// TIA Portal project "AmerikaKamara" (V18)

(* hardware
DEVICE "S7-1200 station_1"  S7-1200 Station
   slot 0: "Rack_0"  S7-1200 Rack  Rack  V1.0
   slot 1: "KamaraFirin"  CPU 1214C DC/DC/DC  6ES7 214-1AG40-0XB0  V4.6
   slot 2: "DI 16/DQ 16x24VDC_1"  6ES7 223-1BL32-0XB0  V2.0
   slot 3: "AQ 4x14BIT_1"  6ES7 232-4HD32-0XB0  V2.1
   slot 3: "CB 1241 (RS485)"  CB 1241 (RS485)  6ES7 241-1CH30-1XB0  V1.0
   slot 4: "AI 4xTC_1"  SM 1231 AI4 x TC  6ES7 231-5QD32-0XB0  V2.0
*)

// ===== PLC "KamaraFirin"  CPU 1214C DC/DC/DC =====

VAR_GLOBAL   // PLC tag table "Default tag table"
   "StartButon" AT %I0.1 : Bool;
   "StopButon" AT %I0.4 : Bool;
   "PompaInvArıza" AT %I0.2 : Bool;
   "ArabaInvArıza" AT %I0.3 : Bool;
   "Tcouple 1" AT %IW128 : Int;
   "Tcouple 1y" AT %IW130 : Int;
   "Tcouple 2" AT %IW132 : Int;
   "Tcouple 2y" AT %IW134 : Int;
   "Damper 1" AT %QW112 : Int;
   "Damper 2" AT %QW114 : Int;
   "Damper 3" AT %QW116 : Int;
   "Damper 4" AT %QW118 : Int;
   "1KapıAcık" AT %I2.0 : Bool;
   "1KapıKapalı" AT %I2.1 : Bool;
   "1KapıYukarda" AT %I2.3 : Bool;
   "1KapıAsagıda" AT %I2.2 : Bool;
   "2KapıAcık" AT %I2.4 : Bool;
   "2KapıKapalı" AT %I2.5 : Bool;
   "2KapıYukarda" AT %I2.7 : Bool;
   "2KapıAsagıda" AT %I2.6 : Bool;
   "1GrupKontaktör" AT %Q2.0 : Bool;
   "1GrupSSR" AT %Q2.1 : Bool;
   "2GrupKontaktör" AT %Q2.4 : Bool;
   "2GrupSSR" AT %Q2.5 : Bool;
   "1KapıAc" AT %Q3.0 : Bool;
   "1KapıKapat" AT %Q3.1 : Bool;
   "1KapıAsagı" AT %Q3.2 : Bool;
   "1KapıYukarı" AT %Q3.3 : Bool;
   "2KapıAc" AT %Q3.4 : Bool;
   "2KapıKapat" AT %Q3.5 : Bool;
   "2KapıAsagı" AT %Q3.6 : Bool;
   "2KapıYukarı" AT %Q3.7 : Bool;
   "AcilStopPano" AT %I0.0 : Bool;
   "HidrolikInverterError" AT %I1.5 : Bool;
   "StartLamba" AT %Q0.0 : Bool;
   "StopLamba" AT %Q0.1 : Bool;
   "HidrolikPompaStart" AT %Q0.2 : Bool;
   "AnaTahliyeValf" AT %Q0.3 : Bool;
   "AcilRöle" AT %Q0.5 : Bool;
   "KırmızıIkaz" AT %Q0.6 : Bool;
   "SarıIkaz" AT %Q0.7 : Bool;
   "YesılIkaz" AT %Q1.0 : Bool;
   "Sıren" AT %Q1.1 : Bool;
   "Emergency" AT %M10.1 : Bool;
   "Error" AT %M10.0 : Bool;
   "currentTemp1Raw" AT %MD100 : Real;
   "currentTemp1" AT %MD104 : Real;
   "SetTimeSnRaw" AT %MD108 : DInt;
   "SetTime" AT %MD112 : Real;
   "SetTemp1Real" AT %MD116 : Real;
   "Ramp1Temp" AT %MD120 : Real;
   "Clock_Byte" AT %MB0 : Byte;
   "Clock_10Hz" AT %M0.0 : Bool;
   "Clock_5Hz" AT %M0.1 : Bool;
   "Clock_2.5Hz" AT %M0.2 : Bool;
   "Clock_2Hz" AT %M0.3 : Bool;
   "Clock_1.25Hz" AT %M0.4 : Bool;
   "Clock_1Hz" AT %M0.5 : Bool;
   "Clock_0.625Hz" AT %M0.6 : Bool;
   "Clock_0.5Hz" AT %M0.7 : Bool;
   "ElapsedSecond" AT %MD124 : Real;
   "elapsed-ramp1" AT %MD128 : Real;
   "StartProcess" AT %M50.0 : Bool;
   "gpwmtimeret1" AT %MD184 : Time;
   "trigclk1" AT %M30.4 : Bool;
   "trigq1" AT %M30.5 : Bool;
   "pwmtimerun1" AT %M30.6 : Bool;
   "pidout1" AT %MD156 : DInt;
   "pidout/20-1" AT %MD188 : UDInt;
   "pidouttime1" AT %MD192 : DWord;
   "currentTemp2Raw" AT %MD160 : Real;
   "currentTemp2" AT %MD164 : Real;
   "SetTemp2Real" AT %MD168 : Real;
   "Ramp2Temp" AT %MD172 : Real;
   "elapsed-ramp2" AT %MD176 : Real;
   "pidout2" AT %MD180 : DInt;
   "trigclk2" AT %M31.0 : Bool;
   "trigq2" AT %M31.1 : Bool;
   "pwmtimerun2" AT %M31.2 : Bool;
   "gpwmtimeret2" AT %MD196 : Time;
   "pidout/20-2" AT %MD200 : UDInt;
   "pidouttime2" AT %MD204 : DWord;
   "Tc1Fark" AT %MD132 : DWord;
   "Tc2Fark" AT %MD136 : DWord;
   "Tc1FarkHata" AT %M30.0 : Bool;
   "Tc2FarkHata" AT %M30.1 : Bool;
   "StepBitti" AT %M30.2 : Bool;
   "StepBittiTrig" AT %M30.3 : Bool;
   "tc1Okunan/10" AT %MD144 : DWord;
   "tc1YOkunan/10" AT %MD148 : DWord;
   "tc2Okunan/10" AT %MD152 : DWord;
   "tc2YOkunan/10" AT %MD140 : DWord;
   "Group2Enable" AT %M20.2 : Bool;
   "Group1Enable" AT %M20.0 : Bool;
   "elapsedTimeTrigClk" AT %M5.0 : Bool;
   "elapsedTimeTrigQ" AT %M5.1 : Bool;
   "startbutonBit" AT %M5.2 : Bool;
   "stopbutonBit" AT %M5.3 : Bool;
   "pidSetTempFark_Q" AT %M5.5 : Bool;
   "baslangicTemp2" AT %MD208 : Real;
   "pidSetTempFark2_Q" AT %M5.6 : Bool;
   "pidSetTemp2" AT %MD212 : Real;
   "baslangicTemp1" AT %MD216 : Real;
   "pidSetTemp1" AT %MD220 : Real;
   "modbusStart" AT %M60.0 : Bool;
   "MBLoadDone" AT %M60.1 : Bool;
   "FrekansCarpilmis" AT %MW224 : UInt;
   "System_Byte" AT %MB1 : Byte;
   "FirstScan" AT %M1.0 : Bool;
   "DiagStatusUpdate" AT %M1.1 : Bool;
   "AlwaysTRUE" AT %M1.2 : Bool;
   "AlwaysFALSE" AT %M1.3 : Bool;
   "ModbusStartScan" AT %M2.0 : Bool;
   "HidrolikBitGeldi" AT %M2.2 : Bool;
   "FrekansYazDone" AT %M60.2 : Bool;
   "KapiAcMinTempError" AT %M350.0 : Bool;
   "DMP1Norm" AT %MD244 : Real;
   "DMP1Scale" AT %MD248 : DWord;
   "DMP2Norm" AT %MD252 : DWord;
   "DMP2Scale" AT %MD256 : DWord;
   "DMP3Norm" AT %MD260 : DWord;
   "DMP3Scale" AT %MD264 : DWord;
   "DMP4Norm" AT %MD268 : DWord;
   "DMP4Scale" AT %MD272 : DWord;
   "HidrolikBit" AT %M400.0 : Bool;
   "akim1Done" AT %M60.4 : Bool;
   "akim2Set" AT %M60.5 : Bool;
   "akim2Done" AT %M60.6 : Bool;
   "akim3Set" AT %M60.7 : Bool;
   "akim1Set" AT %M60.3 : Bool;
   "akim3Done" AT %M61.0 : Bool;
   "akim4Set" AT %M61.1 : Bool;
   "akim4Done" AT %M61.2 : Bool;
   "akim5Set" AT %M61.3 : Bool;
   "akim5Done" AT %M61.4 : Bool;
   "akim6Set" AT %M61.5 : Bool;
   "akim6Done" AT %M61.6 : Bool;
   "HidrolikDelay" AT %MD300 : Time;
   "Tag_1" AT %MD304 : Real;
   "Tag_2" AT %MD308 : DWord;
   "1akim1-2fark" AT %MD312 : DInt;
   "1akim1-2hata" AT %M70.0 : Bool;
   "1akim1-3hata" AT %M70.1 : Bool;
   "1akim1-3fark" AT %MD316 : DInt;
   "1akim2-3fark" AT %MD320 : DInt;
   "1akim2-3hata" AT %M70.2 : Bool;
   "2akim1-2hata" AT %M70.3 : Bool;
   "2akim1-2fark" AT %MD324 : DInt;
   "2akim2-3hata" AT %M70.4 : Bool;
   "2akim1-3fark" AT %MD328 : DInt;
   "2akim2-3hata(1)" AT %M70.5 : Bool;
   "2akim2-3fark" AT %MD332 : DInt;
   "Tag_3" AT %M80.0 : Bool;
   "Reset" AT %M90.0 : Bool;
   "Tag_4" AT %M80.5 : Bool;
   "Tag_5" AT %M5.7 : Bool;
   "kapiacmintemp1" AT %M6.0 : Bool;
   "kapiacmintemp2" AT %M6.1 : Bool;
   "sirenTrigQ" AT %M50.1 : Bool;
   "sirenSet" AT %M50.2 : Bool;
   "kapidelay" AT %MD276 : Time;
   "pompaCalisiyor" AT %M2.3 : Bool;
   "hidrolikdusenkenar" AT %M2.4 : Bool;
END_VAR

DATA_BLOCK "PcdenOkunacak"   // DB2
{ S7_Optimized_Access := 'FALSE' }
VERSION : 0.1
   VAR
      Door1Close : Bool;
      Door1Open : Bool;
      Door1Down : Bool;
      Door1Up : Bool;
      Door2Close : Bool;
      Door2Open : Bool;
      Door2Down : Bool;
      Door2Up : Bool;
      Error : Bool;
      EmergencyPano : Bool;
      HidrolikInveterError : Bool;
      Tc1hata : Bool;
      Tc2Hata : Bool;
      Tc1 : DInt;
      "Tc1.2" : DInt;
      Tc2 : DInt;
      "Tc2.2" : DInt;
      Group1Current : DInt;
      Group2Current : DInt;
      Damper1 : DInt;
      Damper2 : DInt;
      Damper3 : DInt;
      Damper4 : DInt;
      "Step" : DInt;
      butonTime : DInt;
      totalElapsedSec : DInt;
      FirinDurum : Bool;
      butonBasmaTime : Time := T#5S;
      veriGeldi : Bool;
      KapiAcMinTempError : Bool;
      Akim1_1 : Real;
      Akim1_2 : Real;
      Akim1_3 : Real;
      Akim2_1 : Real;
      Akim2_2 : Real;
      Akim2_3 : Real;
      MbLoadError : Bool;
      MbFrekansError : Bool;
      MbAkim1_1Error : Bool;
      MbAkim1_2Error : Bool;
      MbAkim1_3Error : Bool;
      MbAkim2_1Error : Bool;
      MbAkim2_2Error : Bool;
      MbAkim2_3Error : Bool;
      Akim1_1h : Real;
      Akim1_2h : Real;
      Akim1_3h : Real;
      Akim2_1h : Real;
      Akim2_2h : Real;
      Akim2_3h : Real;
      Akim1Ort : DInt;
      Akim2Ort : DInt;
      rezistansError : Bool;
      receteTamam : Bool;
      kapiacildi : Bool;
      Error_1 : Bool;
      siren : Bool;
      elapsedTime : DInt;
      tc1Set : DInt;
      Tc2Set : DInt;
   END_VAR
BEGIN
END_DATA_BLOCK

DATA_BLOCK "PcdenYazilacak"   // DB3
{ S7_Optimized_Access := 'FALSE' }
VERSION : 0.1
   VAR
      Door1Close : Bool;
      Door1Open : Bool;
      Door1Down : Bool;
      Door1Up : Bool;
      Door2Close : Bool;
      Door2Open : Bool;
      Door2Down : Bool;
      Door2Up : Bool;
      SetTemp1 : DInt;
      SetTime : DInt;
      SetTemp2 : DInt;
      Group1Current : DInt;
      Group2Current : DInt;
      Damper1 : DInt;
      Damper2 : DInt;
      Damper3 : DInt;
      Damper4 : DInt;
      TcFarkHata : DInt := 20;
      Group1Run : Bool;
      Group2Run : Bool;
      G1VeriGeldi : Bool;
      G2VeriGeldi : Bool;
      Reset : Bool;
      receteTamam : Bool;
      butonBasmaTime : Time := T#5S;
      SürücüFrekans : Int := 50;
      frekansYaz : Bool;
      sirensustur : Bool;
      MinTemp : DInt := 500;
      ComDelay : Time := T#1s;
      akimFark : DInt := 15;
      adimsayisi : DInt;
   END_VAR
BEGIN
END_DATA_BLOCK

DATA_BLOCK "Group1Control_DB"   // DB6
{ S7_Optimized_Access := 'TRUE' }
VERSION : 0.1
// stored: InstanceOfName Group1Control
"Group1Control"
BEGIN
END_DATA_BLOCK

DATA_BLOCK "Group2Control_DB"   // DB8
{ S7_Optimized_Access := 'TRUE' }
VERSION : 0.1
// stored: InstanceOfName Group2Control
"Group2Control"
BEGIN
END_DATA_BLOCK

// folder: System blocks/Program resources

DATA_BLOCK "ResetTimer"   // DB1
{ S7_Optimized_Access := 'TRUE' }
AUTHOR : Simatic
FAMILY : IEC
NAME : IEC_TMR
VERSION : 1.0
// stored: InstanceOfName IEC_TIMER
"IEC_TIMER"
BEGIN
END_DATA_BLOCK

DATA_BLOCK "IslemBittiTimer"   // DB4
{ S7_Optimized_Access := 'TRUE' }
AUTHOR : Simatic
FAMILY : IEC
NAME : IEC_TMR
VERSION : 1.0
// stored: InstanceOfName IEC_TIMER
"IEC_TIMER"
BEGIN
END_DATA_BLOCK

DATA_BLOCK "Group1PwmTimer"   // DB10
{ S7_Optimized_Access := 'TRUE' }
AUTHOR : Simatic
FAMILY : IEC
NAME : IEC_TMR
VERSION : 1.0
// stored: InstanceOfName IEC_TIMER
"IEC_TIMER"
BEGIN
END_DATA_BLOCK

DATA_BLOCK "Group2PwmTimer"   // DB12
{ S7_Optimized_Access := 'TRUE' }
AUTHOR : Simatic
FAMILY : IEC
NAME : IEC_TMR
VERSION : 1.0
// stored: InstanceOfName IEC_TIMER
"IEC_TIMER"
BEGIN
END_DATA_BLOCK

DATA_BLOCK "AnaValfGecikme"   // DB19
{ S7_Optimized_Access := 'TRUE' }
AUTHOR : Simatic
FAMILY : IEC
NAME : IEC_TMR
VERSION : 1.0
// stored: InstanceOfName IEC_TIMER
"IEC_TIMER"
BEGIN
END_DATA_BLOCK

DATA_BLOCK "PompaGecikme"   // DB20
{ S7_Optimized_Access := 'TRUE' }
AUTHOR : Simatic
FAMILY : IEC
NAME : IEC_TMR
VERSION : 1.0
// stored: InstanceOfName IEC_TIMER
"IEC_TIMER"
BEGIN
END_DATA_BLOCK

DATA_BLOCK "MBCycleDelay"   // DB21
{ S7_Optimized_Access := 'TRUE' }
AUTHOR : Simatic
FAMILY : IEC
NAME : IEC_TMR
VERSION : 1.0
// stored: InstanceOfName IEC_TIMER
"IEC_TIMER"
BEGIN
END_DATA_BLOCK

DATA_BLOCK "akim1TM"   // DB22
{ S7_Optimized_Access := 'TRUE' }
AUTHOR : Simatic
FAMILY : IEC
NAME : IEC_TMR
VERSION : 1.0
// stored: InstanceOfName IEC_TIMER
"IEC_TIMER"
BEGIN
END_DATA_BLOCK

DATA_BLOCK "akim2TM"   // DB23
{ S7_Optimized_Access := 'TRUE' }
AUTHOR : Simatic
FAMILY : IEC
NAME : IEC_TMR
VERSION : 1.0
// stored: InstanceOfName IEC_TIMER
"IEC_TIMER"
BEGIN
END_DATA_BLOCK

DATA_BLOCK "akim3TM"   // DB24
{ S7_Optimized_Access := 'TRUE' }
AUTHOR : Simatic
FAMILY : IEC
NAME : IEC_TMR
VERSION : 1.0
// stored: InstanceOfName IEC_TIMER
"IEC_TIMER"
BEGIN
END_DATA_BLOCK

DATA_BLOCK "akim4TM"   // DB25
{ S7_Optimized_Access := 'TRUE' }
AUTHOR : Simatic
FAMILY : IEC
NAME : IEC_TMR
VERSION : 1.0
// stored: InstanceOfName IEC_TIMER
"IEC_TIMER"
BEGIN
END_DATA_BLOCK

DATA_BLOCK "akim5TM"   // DB26
{ S7_Optimized_Access := 'TRUE' }
AUTHOR : Simatic
FAMILY : IEC
NAME : IEC_TMR
VERSION : 1.0
// stored: InstanceOfName IEC_TIMER
"IEC_TIMER"
BEGIN
END_DATA_BLOCK

DATA_BLOCK "akim6TM"   // DB27
{ S7_Optimized_Access := 'TRUE' }
AUTHOR : Simatic
FAMILY : IEC
NAME : IEC_TMR
VERSION : 1.0
// stored: InstanceOfName IEC_TIMER
"IEC_TIMER"
BEGIN
END_DATA_BLOCK

DATA_BLOCK "IEC_Timer_0_DB"   // DB28
{ S7_Optimized_Access := 'TRUE' }
AUTHOR : Simatic
FAMILY : IEC
NAME : IEC_TMR
VERSION : 1.0
// stored: InstanceOfName IEC_TIMER
"IEC_TIMER"
BEGIN
END_DATA_BLOCK

DATA_BLOCK "rezistansErrorTmr"   // DB29
{ S7_Optimized_Access := 'TRUE' }
AUTHOR : Simatic
FAMILY : IEC
NAME : IEC_TMR
VERSION : 1.0
// stored: InstanceOfName IEC_TIMER
"IEC_TIMER"
BEGIN
END_DATA_BLOCK

DATA_BLOCK "IEC_Timer_0_DB_1"   // DB30
{ S7_Optimized_Access := 'TRUE' }
AUTHOR : Simatic
FAMILY : IEC
NAME : IEC_TMR
VERSION : 1.0
// stored: InstanceOfName IEC_TIMER
"IEC_TIMER"
BEGIN
END_DATA_BLOCK

DATA_BLOCK "IEC_Timer_0_DB_2"   // DB31
{ S7_Optimized_Access := 'TRUE' }
AUTHOR : Simatic
FAMILY : IEC
NAME : IEC_TMR
VERSION : 1.0
// stored: InstanceOfName IEC_TIMER
"IEC_TIMER"
BEGIN
END_DATA_BLOCK

DATA_BLOCK "ErrorStopDelay"   // DB32
{ S7_Optimized_Access := 'TRUE' }
AUTHOR : Simatic
FAMILY : IEC
NAME : IEC_TMR
VERSION : 1.0
// stored: InstanceOfName IEC_TIMER
"IEC_TIMER"
BEGIN
END_DATA_BLOCK

DATA_BLOCK "tcErrorDelay"   // DB33
{ S7_Optimized_Access := 'TRUE' }
AUTHOR : Simatic
FAMILY : IEC
NAME : IEC_TMR
VERSION : 1.0
// stored: InstanceOfName IEC_TIMER
"IEC_TIMER"
BEGIN
END_DATA_BLOCK

DATA_BLOCK "kapi1acikdelay"   // DB35
{ S7_Optimized_Access := 'TRUE' }
AUTHOR : Simatic
FAMILY : IEC
NAME : IEC_TMR
VERSION : 1.0
// stored: InstanceOfName IEC_TIMER
"IEC_TIMER"
BEGIN
END_DATA_BLOCK

DATA_BLOCK "kapi1kapalidelay"   // DB36
{ S7_Optimized_Access := 'TRUE' }
AUTHOR : Simatic
FAMILY : IEC
NAME : IEC_TMR
VERSION : 1.0
// stored: InstanceOfName IEC_TIMER
"IEC_TIMER"
BEGIN
END_DATA_BLOCK

DATA_BLOCK "kapi2acikdelay"   // DB37
{ S7_Optimized_Access := 'TRUE' }
AUTHOR : Simatic
FAMILY : IEC
NAME : IEC_TMR
VERSION : 1.0
// stored: InstanceOfName IEC_TIMER
"IEC_TIMER"
BEGIN
END_DATA_BLOCK

DATA_BLOCK "kapi2kapalidelay"   // DB38
{ S7_Optimized_Access := 'TRUE' }
AUTHOR : Simatic
FAMILY : IEC
NAME : IEC_TMR
VERSION : 1.0
// stored: InstanceOfName IEC_TIMER
"IEC_TIMER"
BEGIN
END_DATA_BLOCK

DATA_BLOCK "sirenSusturtmr"   // DB39
{ S7_Optimized_Access := 'TRUE' }
AUTHOR : Simatic
FAMILY : IEC
NAME : IEC_TMR
VERSION : 1.0
// stored: InstanceOfName IEC_TIMER
"IEC_TIMER"
BEGIN
END_DATA_BLOCK

// folder: (top level)

FUNCTION_BLOCK "Group1Control"   // FB1, LAD
{ S7_Optimized_Access := 'TRUE' }
VERSION : 0.1
   VAR_INPUT
      "m20.0" : Bool;
   END_VAR
BEGIN

REGION Network 1: Group 1 Heating
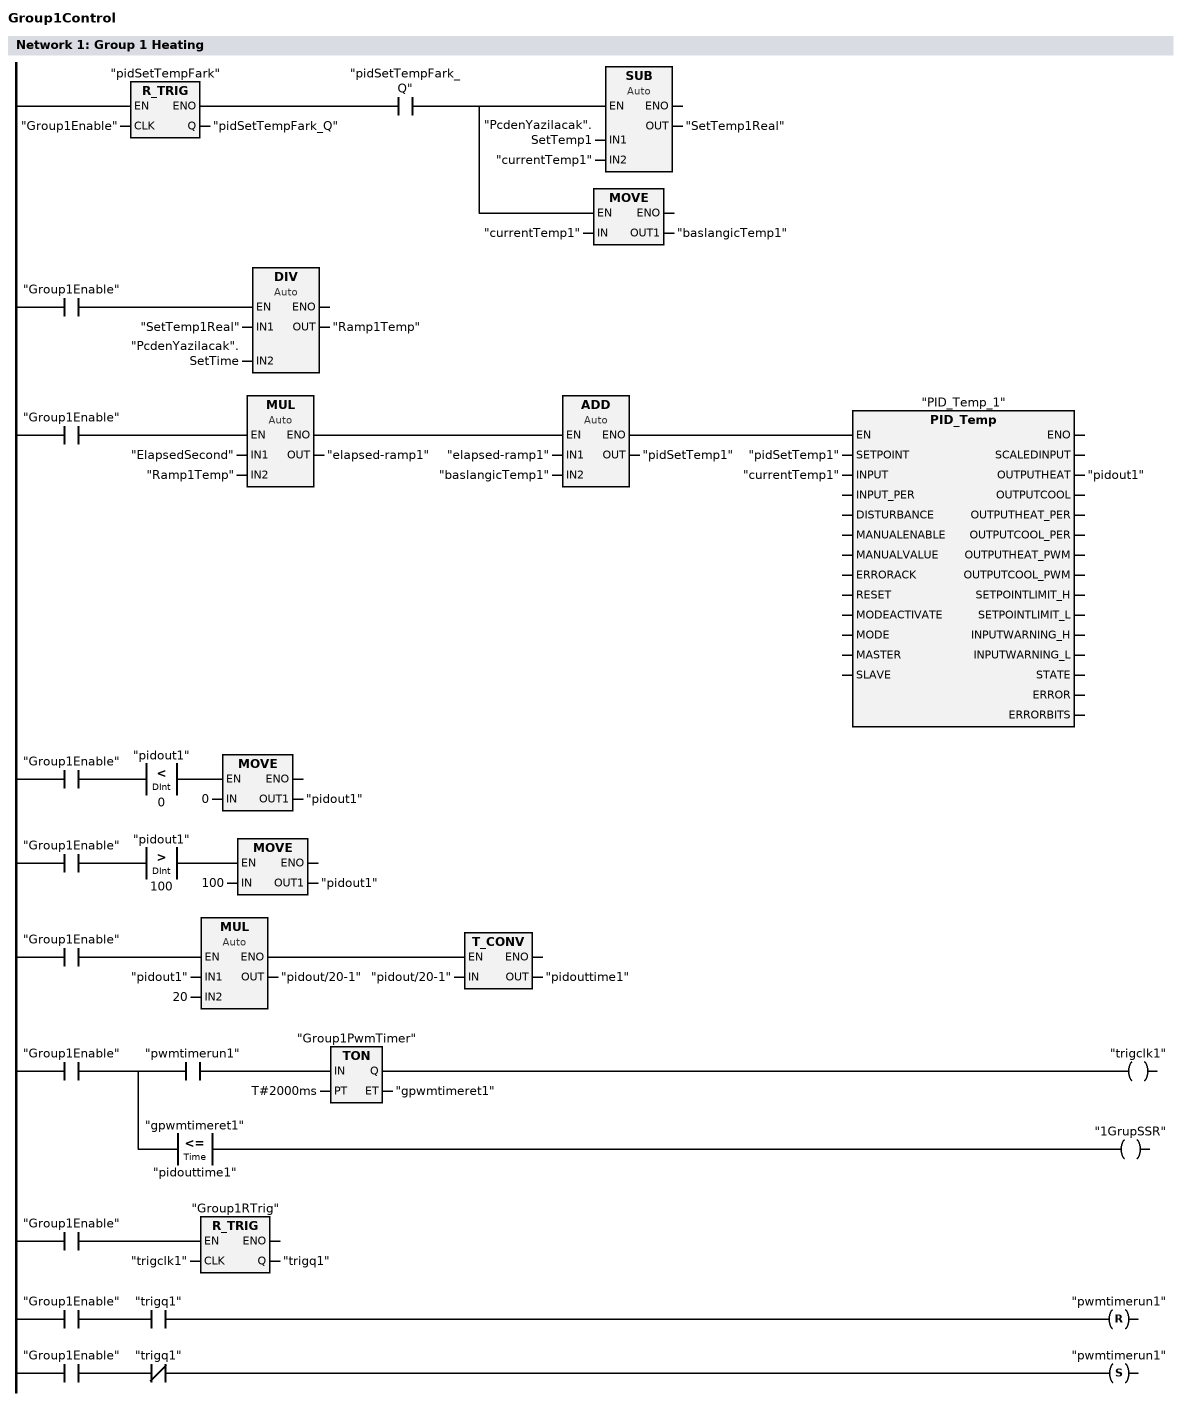
   // ENO of a box is taken as its EN; it also drops when the box reports an error
   "pidSetTempFark"(CLK := "Group1Enable", Q => "pidSetTempFark_Q");   // R_TRIG
   IF "pidSetTempFark_Q" THEN
       "SetTemp1Real" := "PcdenYazilacak".SetTemp1 - "currentTemp1";
       "baslangicTemp1" := "currentTemp1";
   END_IF;
   IF "Group1Enable" THEN
       "Ramp1Temp" := "SetTemp1Real" / "PcdenYazilacak".SetTime;
       "elapsed-ramp1" := "ElapsedSecond" * "Ramp1Temp";
       "pidSetTemp1" := "elapsed-ramp1" + "baslangicTemp1";
       "PID_Temp_1"(Setpoint := "pidSetTemp1", Input := "currentTemp1", OutputHeat => "pidout1");   // PID_Temp
   END_IF;
   IF "Group1Enable" AND ("pidout1" < 0) THEN "pidout1" := 0; END_IF;
   IF "Group1Enable" AND ("pidout1" > 100) THEN "pidout1" := 100; END_IF;
   IF "Group1Enable" THEN
       "pidout/20-1" := "pidout1" * 20;
       "pidouttime1" := T_CONV(IN := "pidout/20-1");
   END_IF;
   "Group1PwmTimer".TON(IN := "Group1Enable" AND "pwmtimerun1", PT := T#2000ms, ET => "gpwmtimeret1");
   "trigclk1" := "Group1PwmTimer".Q;
   "1GrupSSR" := "Group1Enable" AND ("gpwmtimeret1" <= "pidouttime1");
   IF "Group1Enable" THEN
       "Group1RTrig"(CLK := "trigclk1", Q => "trigq1");   // R_TRIG
   END_IF;
   IF "Group1Enable" AND "trigq1" THEN "pwmtimerun1" := FALSE; END_IF;
   IF "Group1Enable" AND NOT "trigq1" THEN "pwmtimerun1" := TRUE; END_IF;
END_REGION
END_FUNCTION_BLOCK

FUNCTION_BLOCK "Group2Control"   // FB2, LAD
{ S7_Optimized_Access := 'TRUE' }
VERSION : 0.1
   VAR_INPUT
      "m20.2" : Bool;
   END_VAR
BEGIN

REGION Network 1
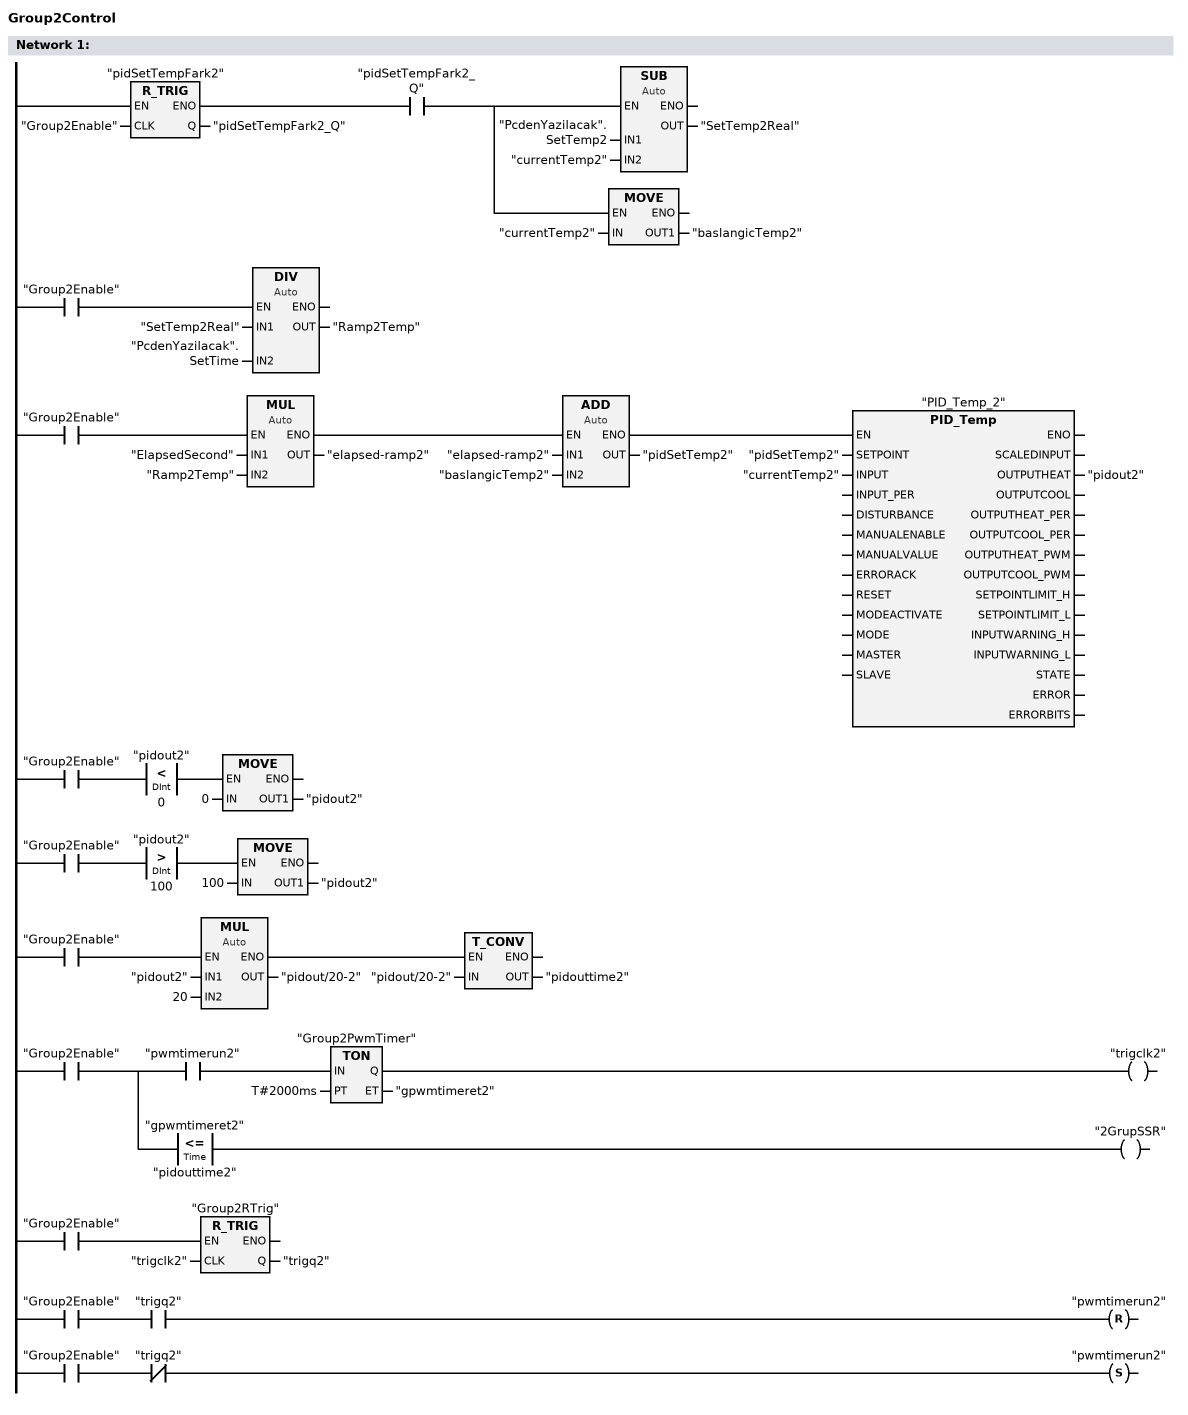
   // ENO of a box is taken as its EN; it also drops when the box reports an error
   "pidSetTempFark2"(CLK := "Group2Enable", Q => "pidSetTempFark2_Q");   // R_TRIG
   IF "pidSetTempFark2_Q" THEN
       "SetTemp2Real" := "PcdenYazilacak".SetTemp2 - "currentTemp2";
       "baslangicTemp2" := "currentTemp2";
   END_IF;
   IF "Group2Enable" THEN
       "Ramp2Temp" := "SetTemp2Real" / "PcdenYazilacak".SetTime;
       "elapsed-ramp2" := "ElapsedSecond" * "Ramp2Temp";
       "pidSetTemp2" := "elapsed-ramp2" + "baslangicTemp2";
       "PID_Temp_2"(Setpoint := "pidSetTemp2", Input := "currentTemp2", OutputHeat => "pidout2");   // PID_Temp
   END_IF;
   IF "Group2Enable" AND ("pidout2" < 0) THEN "pidout2" := 0; END_IF;
   IF "Group2Enable" AND ("pidout2" > 100) THEN "pidout2" := 100; END_IF;
   IF "Group2Enable" THEN
       "pidout/20-2" := "pidout2" * 20;
       "pidouttime2" := T_CONV(IN := "pidout/20-2");
   END_IF;
   "Group2PwmTimer".TON(IN := "Group2Enable" AND "pwmtimerun2", PT := T#2000ms, ET => "gpwmtimeret2");
   "trigclk2" := "Group2PwmTimer".Q;
   "2GrupSSR" := "Group2Enable" AND ("gpwmtimeret2" <= "pidouttime2");
   IF "Group2Enable" THEN
       "Group2RTrig"(CLK := "trigclk2", Q => "trigq2");   // R_TRIG
   END_IF;
   IF "Group2Enable" AND "trigq2" THEN "pwmtimerun2" := FALSE; END_IF;
   IF "Group2Enable" AND NOT "trigq2" THEN "pwmtimerun2" := TRUE; END_IF;
END_REGION
END_FUNCTION_BLOCK

ORGANIZATION_BLOCK "Main"   // OB1, LAD, ProgramCycle
TITLE = "Main Program Sweep (Cycle)"
{ S7_Optimized_Access := 'TRUE' }
VERSION : 0.1
   VAR_INPUT
      Initial_Call : Bool;   // Initial call of this OB
      Remanence : Bool;   // =True, if remanent data are available
   END_VAR
   VAR_TEMP   // added for the SCL form of the ladder/FBD networks
      _w1 : Bool;
      _w2 : Bool;
      _w3 : Bool;
      _w4 : Bool;
      _w5 : Bool;
      _w6 : Bool;
      _w7 : Bool;
   END_VAR
BEGIN

REGION Network 1: startProcess
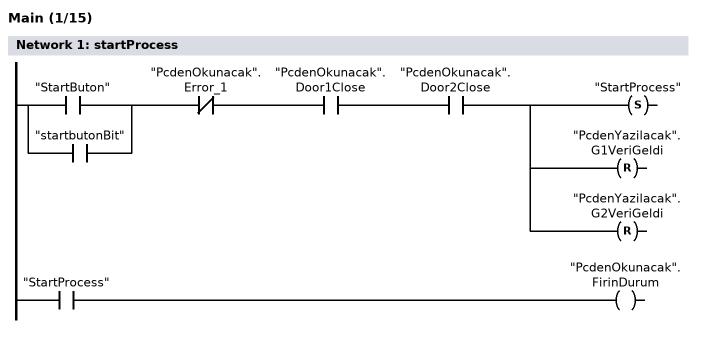
   RUNG wire#powerrail
      Contact( "StartButon" )
      wire#w1
      I_Contact( "PcdenOkunacak".Error_1 )
      Contact( "PcdenOkunacak".Door1Close )
      Contact( "PcdenOkunacak".Door2Close )
      wire#w2
      S_Coil( "StartProcess" )
   END_RUNG
   RUNG wire#powerrail
      Contact( "startbutonBit" )
   END_RUNG wire#w1
   RUNG wire#w2
      R_Coil( "PcdenYazilacak".G1VeriGeldi )
   END_RUNG
   RUNG wire#w2
      R_Coil( "PcdenYazilacak".G2VeriGeldi )
   END_RUNG
   RUNG wire#powerrail
      Contact( "StartProcess" )
      Coil( "PcdenOkunacak".FirinDurum )
   END_RUNG
   // the same network as SCL:
   IF ("StartButon" OR "startbutonBit") AND NOT "PcdenOkunacak".Error_1 AND "PcdenOkunacak".Door1Close AND "PcdenOkunacak".Door2Close THEN
       "StartProcess" := TRUE;
       "PcdenYazilacak".G1VeriGeldi := FALSE;
       "PcdenYazilacak".G2VeriGeldi := FALSE;
   END_IF;
   "PcdenOkunacak".FirinDurum := "StartProcess";
END_REGION

REGION Network 2: Stop and Reset
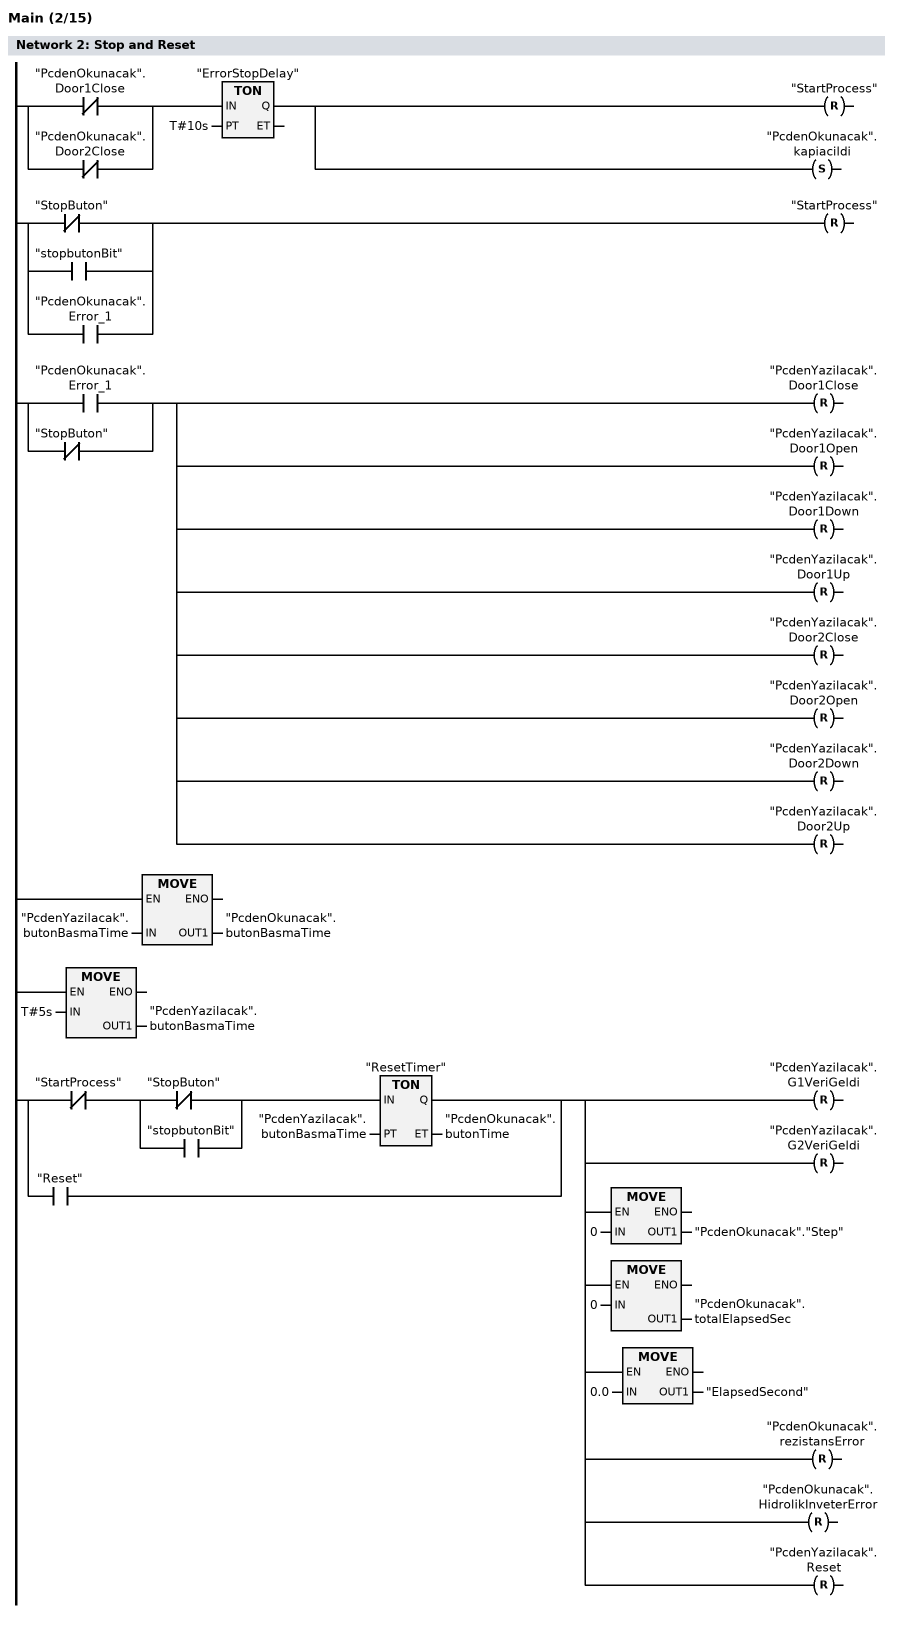
   "ErrorStopDelay".TON(IN := NOT "PcdenOkunacak".Door1Close OR NOT "PcdenOkunacak".Door2Close, PT := T#10s);
   IF "ErrorStopDelay".Q THEN
       "StartProcess" := FALSE;
       "PcdenOkunacak".kapiacildi := TRUE;
   END_IF;
   IF NOT "StopButon" OR "stopbutonBit" OR "PcdenOkunacak".Error_1 THEN "StartProcess" := FALSE; END_IF;
   IF "PcdenOkunacak".Error_1 OR NOT "StopButon" THEN
       "PcdenYazilacak".Door1Close := FALSE;
       "PcdenYazilacak".Door1Open := FALSE;
       "PcdenYazilacak".Door1Down := FALSE;
       "PcdenYazilacak".Door1Up := FALSE;
       "PcdenYazilacak".Door2Close := FALSE;
       "PcdenYazilacak".Door2Open := FALSE;
       "PcdenYazilacak".Door2Down := FALSE;
       "PcdenYazilacak".Door2Up := FALSE;
   END_IF;
   "PcdenOkunacak".butonBasmaTime := "PcdenYazilacak".butonBasmaTime;
   "PcdenYazilacak".butonBasmaTime := T#5s;
   "ResetTimer".TON(IN := NOT "StartProcess" AND (NOT "StopButon" OR "stopbutonBit"),
                    PT := "PcdenYazilacak".butonBasmaTime,
                    ET => "PcdenOkunacak".butonTime);
   IF "ResetTimer".Q OR "Reset" THEN
       "PcdenYazilacak".G1VeriGeldi := FALSE;
       "PcdenYazilacak".G2VeriGeldi := FALSE;
       "PcdenOkunacak"."Step" := 0;
       "PcdenOkunacak".totalElapsedSec := 0;
       "ElapsedSecond" := 0.0;
       "PcdenOkunacak".rezistansError := FALSE;
       "PcdenOkunacak".HidrolikInveterError := FALSE;
       "PcdenYazilacak".Reset := FALSE;
   END_IF;
END_REGION

REGION Network 3: Cycle Step and Time
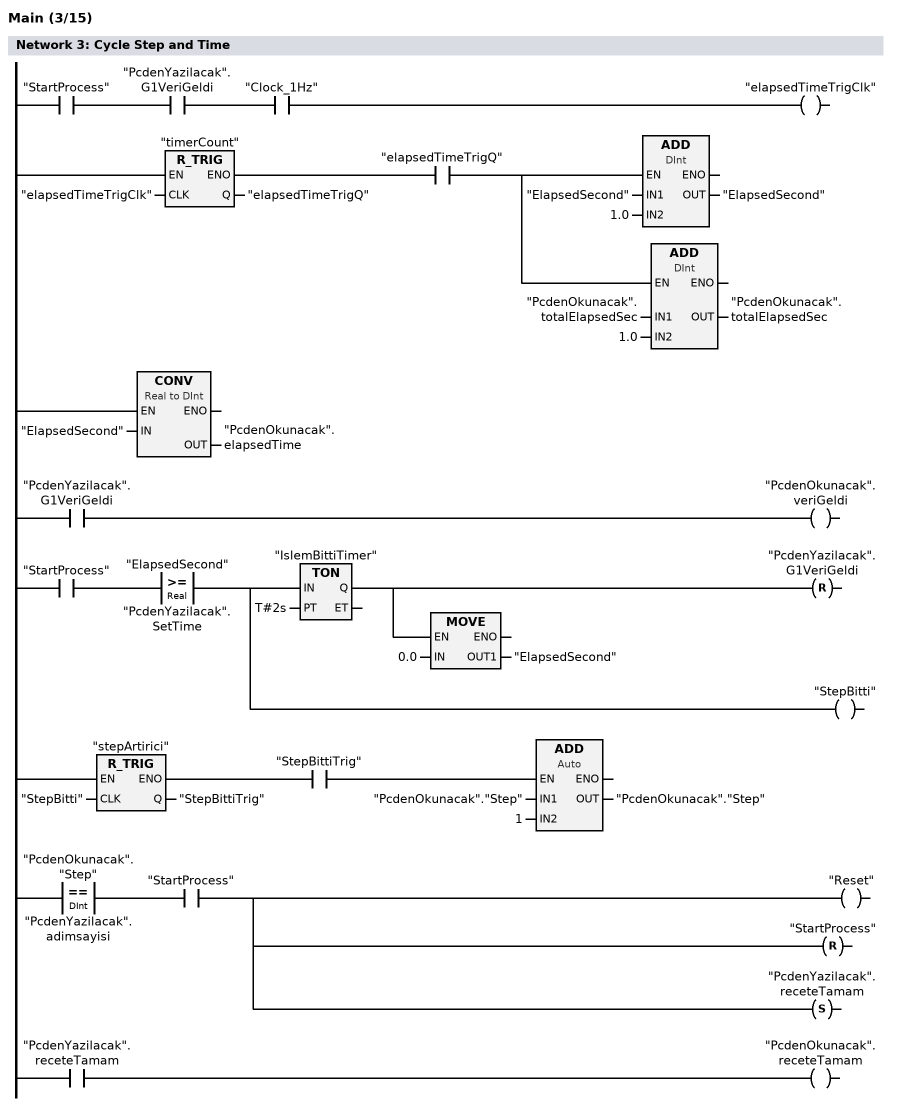
   // ENO of a box is taken as its EN; it also drops when the box reports an error
   "elapsedTimeTrigClk" := "StartProcess" AND "PcdenYazilacak".G1VeriGeldi AND "Clock_1Hz";
   "timerCount"(CLK := "elapsedTimeTrigClk", Q => "elapsedTimeTrigQ");   // R_TRIG
   IF "elapsedTimeTrigQ" THEN
       "ElapsedSecond" := "ElapsedSecond" + 1.0;
       "PcdenOkunacak".totalElapsedSec := "PcdenOkunacak".totalElapsedSec + 1.0;
   END_IF;
   "PcdenOkunacak".elapsedTime := REAL_TO_DINT("ElapsedSecond");
   "PcdenOkunacak".veriGeldi := "PcdenYazilacak".G1VeriGeldi;
   #_w1 := "StartProcess" AND ("ElapsedSecond" >= "PcdenYazilacak".SetTime);
   "IslemBittiTimer".TON(IN := #_w1, PT := T#2s);
   IF "IslemBittiTimer".Q THEN
       "PcdenYazilacak".G1VeriGeldi := FALSE;
       "ElapsedSecond" := 0.0;
   END_IF;
   "StepBitti" := #_w1;
   "stepArtirici"(CLK := "StepBitti", Q => "StepBittiTrig");   // R_TRIG
   IF "StepBittiTrig" THEN "PcdenOkunacak"."Step" := "PcdenOkunacak"."Step" + 1; END_IF;
   "Reset" := ("PcdenOkunacak"."Step" = "PcdenYazilacak".adimsayisi) AND "StartProcess";
   IF "Reset" THEN
       "StartProcess" := FALSE;
       "PcdenYazilacak".receteTamam := TRUE;
   END_IF;
   "PcdenOkunacak".receteTamam := "PcdenYazilacak".receteTamam;
END_REGION

REGION Network 4: Group 1 Heating
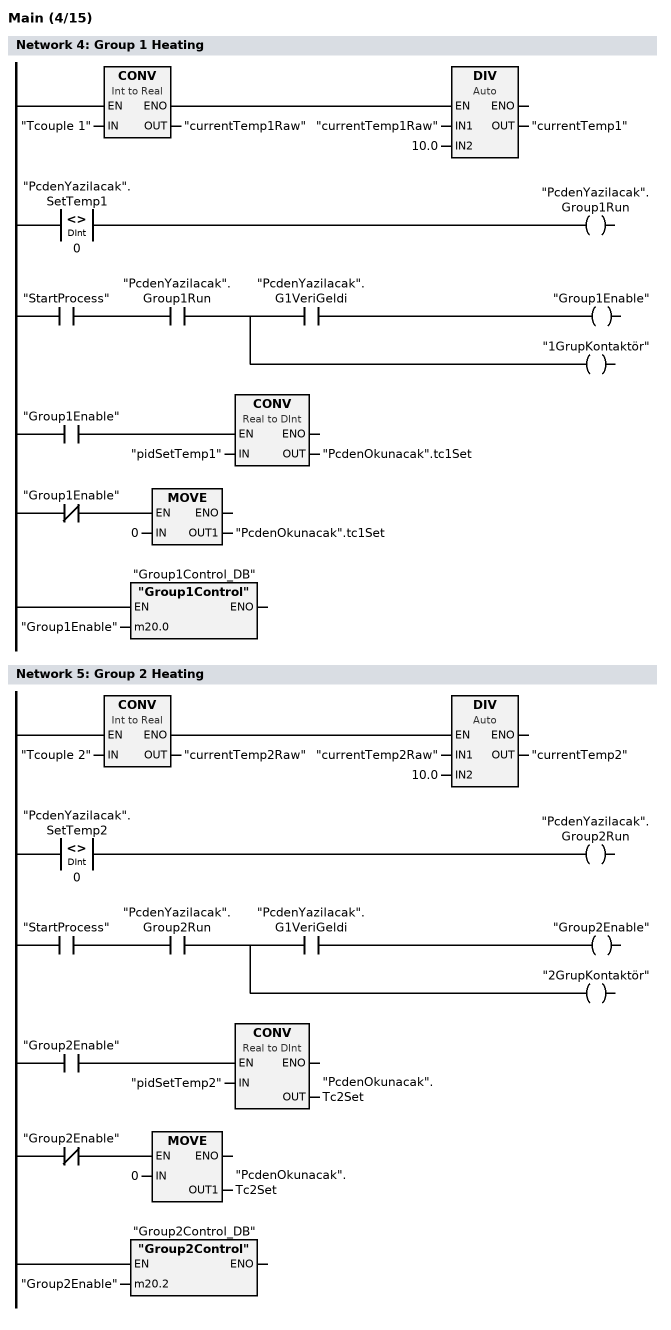
   RUNG wire#powerrail
      { S7_Templates := "[SrcType := Int, DestType := Real]" } Convert(in := "Tcouple 1", out => "currentTemp1Raw")
      Div(in1 := "currentTemp1Raw", in2 := 10.0, out => "currentTemp1")
   END_RUNG
   RUNG wire#powerrail
      { S7_Templates := "SrcType := DInt" } NE_Contact(in1 := "PcdenYazilacak".SetTemp1, in2 := 0)
      Coil( "PcdenYazilacak".Group1Run )
   END_RUNG
   RUNG wire#powerrail
      Contact( "StartProcess" )
      Contact( "PcdenYazilacak".Group1Run )
      wire#w1
      Contact( "PcdenYazilacak".G1VeriGeldi )
      Coil( "Group1Enable" )
   END_RUNG
   RUNG wire#w1
      Coil( "1GrupKontaktör" )
   END_RUNG
   RUNG wire#powerrail
      Contact( "Group1Enable" )
      { S7_Templates := "[SrcType := Real, DestType := DInt]" } Convert(in := "pidSetTemp1", out => "PcdenOkunacak".tc1Set)
   END_RUNG
   RUNG wire#powerrail
      I_Contact( "Group1Enable" )
      Move(in := 0, out1 => "PcdenOkunacak".tc1Set)
   END_RUNG
   RUNG wire#powerrail
      "Group1Control_DB"("m20.0" := "Group1Enable")
   END_RUNG
   // the same network as SCL:
   "currentTemp1Raw" := INT_TO_REAL("Tcouple 1");
   "currentTemp1" := "currentTemp1Raw" / 10.0;
   "PcdenYazilacak".Group1Run := "PcdenYazilacak".SetTemp1 <> 0;
   #_w1 := "StartProcess" AND "PcdenYazilacak".Group1Run;
   "Group1Enable" := #_w1 AND "PcdenYazilacak".G1VeriGeldi;
   "1GrupKontaktör" := #_w1;
   IF "Group1Enable" THEN "PcdenOkunacak".tc1Set := REAL_TO_DINT("pidSetTemp1"); END_IF;
   IF NOT "Group1Enable" THEN "PcdenOkunacak".tc1Set := 0; END_IF;
   "Group1Control_DB"("m20.0" := "Group1Enable");   // "Group1Control"
END_REGION

REGION Network 5: Group 2 Heating
   RUNG wire#powerrail
      { S7_Templates := "[SrcType := Int, DestType := Real]" } Convert(in := "Tcouple 2", out => "currentTemp2Raw")
      Div(in1 := "currentTemp2Raw", in2 := 10.0, out => "currentTemp2")
   END_RUNG
   RUNG wire#powerrail
      { S7_Templates := "SrcType := DInt" } NE_Contact(in1 := "PcdenYazilacak".SetTemp2, in2 := 0)
      Coil( "PcdenYazilacak".Group2Run )
   END_RUNG
   RUNG wire#powerrail
      Contact( "StartProcess" )
      Contact( "PcdenYazilacak".Group2Run )
      wire#w1
      Contact( "PcdenYazilacak".G1VeriGeldi )
      Coil( "Group2Enable" )
   END_RUNG
   RUNG wire#w1
      Coil( "2GrupKontaktör" )
   END_RUNG
   RUNG wire#powerrail
      Contact( "Group2Enable" )
      { S7_Templates := "[SrcType := Real, DestType := DInt]" } Convert(in := "pidSetTemp2", out => "PcdenOkunacak".Tc2Set)
   END_RUNG
   RUNG wire#powerrail
      I_Contact( "Group2Enable" )
      Move(in := 0, out1 => "PcdenOkunacak".Tc2Set)
   END_RUNG
   RUNG wire#powerrail
      "Group2Control_DB"("m20.2" := "Group2Enable")
   END_RUNG
   // the same network as SCL:
   "currentTemp2Raw" := INT_TO_REAL("Tcouple 2");
   "currentTemp2" := "currentTemp2Raw" / 10.0;
   "PcdenYazilacak".Group2Run := "PcdenYazilacak".SetTemp2 <> 0;
   #_w1 := "StartProcess" AND "PcdenYazilacak".Group2Run;
   "Group2Enable" := #_w1 AND "PcdenYazilacak".G1VeriGeldi;
   "2GrupKontaktör" := #_w1;
   IF "Group2Enable" THEN "PcdenOkunacak".Tc2Set := REAL_TO_DINT("pidSetTemp2"); END_IF;
   IF NOT "Group2Enable" THEN "PcdenOkunacak".Tc2Set := 0; END_IF;
   "Group2Control_DB"("m20.2" := "Group2Enable");   // "Group2Control"
END_REGION

REGION Network 6: TCouple
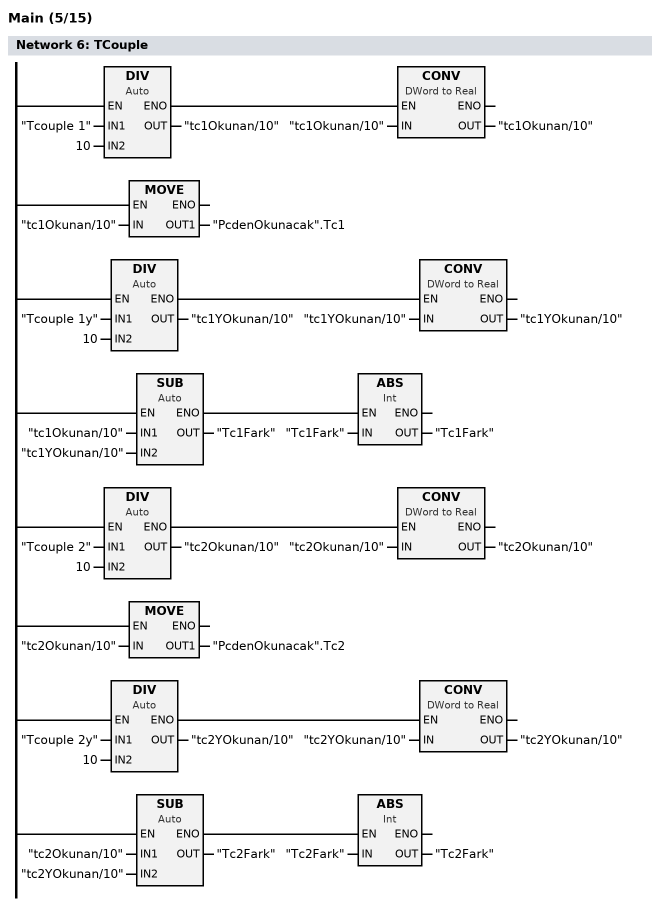
   RUNG wire#powerrail
      Div(in1 := "Tcouple 1", in2 := 10, out => "tc1Okunan/10")
      { S7_Templates := "[SrcType := DWord, DestType := Real]" } Convert(in := "tc1Okunan/10", out => "tc1Okunan/10")
   END_RUNG
   RUNG wire#powerrail
      Move(in := "tc1Okunan/10", out1 => "PcdenOkunacak".Tc1)
   END_RUNG
   RUNG wire#powerrail
      Div(in1 := "Tcouple 1y", in2 := 10, out => "tc1YOkunan/10")
      { S7_Templates := "[SrcType := DWord, DestType := Real]" } Convert(in := "tc1YOkunan/10", out => "tc1YOkunan/10")
   END_RUNG
   RUNG wire#powerrail
      Sub(in1 := "tc1Okunan/10", in2 := "tc1YOkunan/10", out => "Tc1Fark")
      { S7_Templates := "SrcType := Int" } Abs(in := "Tc1Fark", out => "Tc1Fark")
   END_RUNG
   RUNG wire#powerrail
      Div(in1 := "Tcouple 2", in2 := 10, out => "tc2Okunan/10")
      { S7_Templates := "[SrcType := DWord, DestType := Real]" } Convert(in := "tc2Okunan/10", out => "tc2Okunan/10")
   END_RUNG
   RUNG wire#powerrail
      Move(in := "tc2Okunan/10", out1 => "PcdenOkunacak".Tc2)
   END_RUNG
   RUNG wire#powerrail
      Div(in1 := "Tcouple 2y", in2 := 10, out => "tc2YOkunan/10")
      { S7_Templates := "[SrcType := DWord, DestType := Real]" } Convert(in := "tc2YOkunan/10", out => "tc2YOkunan/10")
   END_RUNG
   RUNG wire#powerrail
      Sub(in1 := "tc2Okunan/10", in2 := "tc2YOkunan/10", out => "Tc2Fark")
      { S7_Templates := "SrcType := Int" } Abs(in := "Tc2Fark", out => "Tc2Fark")
   END_RUNG
   // the same network as SCL:
   "tc1Okunan/10" := "Tcouple 1" / 10;
   "tc1Okunan/10" := DWORD_TO_REAL("tc1Okunan/10");
   "PcdenOkunacak".Tc1 := "tc1Okunan/10";
   "tc1YOkunan/10" := "Tcouple 1y" / 10;
   "tc1YOkunan/10" := DWORD_TO_REAL("tc1YOkunan/10");
   "Tc1Fark" := "tc1Okunan/10" - "tc1YOkunan/10";
   "Tc1Fark" := ABS("Tc1Fark");
   "tc2Okunan/10" := "Tcouple 2" / 10;
   "tc2Okunan/10" := DWORD_TO_REAL("tc2Okunan/10");
   "PcdenOkunacak".Tc2 := "tc2Okunan/10";
   "tc2YOkunan/10" := "Tcouple 2y" / 10;
   "tc2YOkunan/10" := DWORD_TO_REAL("tc2YOkunan/10");
   "Tc2Fark" := "tc2Okunan/10" - "tc2YOkunan/10";
   "Tc2Fark" := ABS("Tc2Fark");
END_REGION

REGION Network 7: Emergency
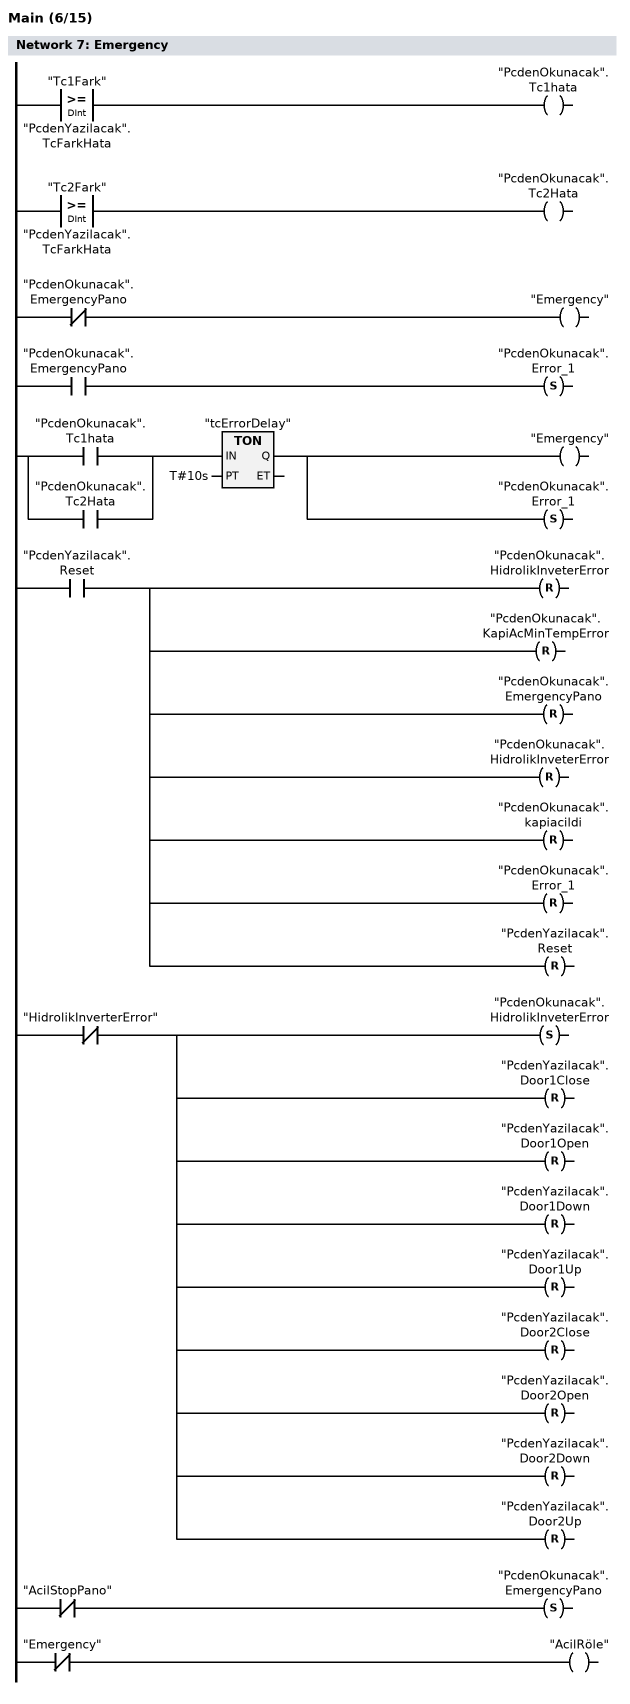
   "PcdenOkunacak".Tc1hata := "Tc1Fark" >= "PcdenYazilacak".TcFarkHata;
   "PcdenOkunacak".Tc2Hata := "Tc2Fark" >= "PcdenYazilacak".TcFarkHata;
   "Emergency" := NOT "PcdenOkunacak".EmergencyPano;
   IF "PcdenOkunacak".EmergencyPano THEN "PcdenOkunacak".Error_1 := TRUE; END_IF;
   "tcErrorDelay".TON(IN := "PcdenOkunacak".Tc1hata OR "PcdenOkunacak".Tc2Hata, PT := T#10s);
   "Emergency" := "tcErrorDelay".Q;
   IF "tcErrorDelay".Q THEN "PcdenOkunacak".Error_1 := TRUE; END_IF;
   IF "PcdenYazilacak".Reset THEN
       "PcdenOkunacak".HidrolikInveterError := FALSE;
       "PcdenOkunacak".KapiAcMinTempError := FALSE;
       "PcdenOkunacak".EmergencyPano := FALSE;
       "PcdenOkunacak".HidrolikInveterError := FALSE;
       "PcdenOkunacak".kapiacildi := FALSE;
       "PcdenOkunacak".Error_1 := FALSE;
       "PcdenYazilacak".Reset := FALSE;
   END_IF;
   IF NOT "HidrolikInverterError" THEN
       "PcdenOkunacak".HidrolikInveterError := TRUE;
       "PcdenYazilacak".Door1Close := FALSE;
       "PcdenYazilacak".Door1Open := FALSE;
       "PcdenYazilacak".Door1Down := FALSE;
       "PcdenYazilacak".Door1Up := FALSE;
       "PcdenYazilacak".Door2Close := FALSE;
       "PcdenYazilacak".Door2Open := FALSE;
       "PcdenYazilacak".Door2Down := FALSE;
       "PcdenYazilacak".Door2Up := FALSE;
   END_IF;
   IF NOT "AcilStopPano" THEN "PcdenOkunacak".EmergencyPano := TRUE; END_IF;
   "AcilRöle" := NOT "Emergency";
END_REGION

REGION Network 8: Door Inputs
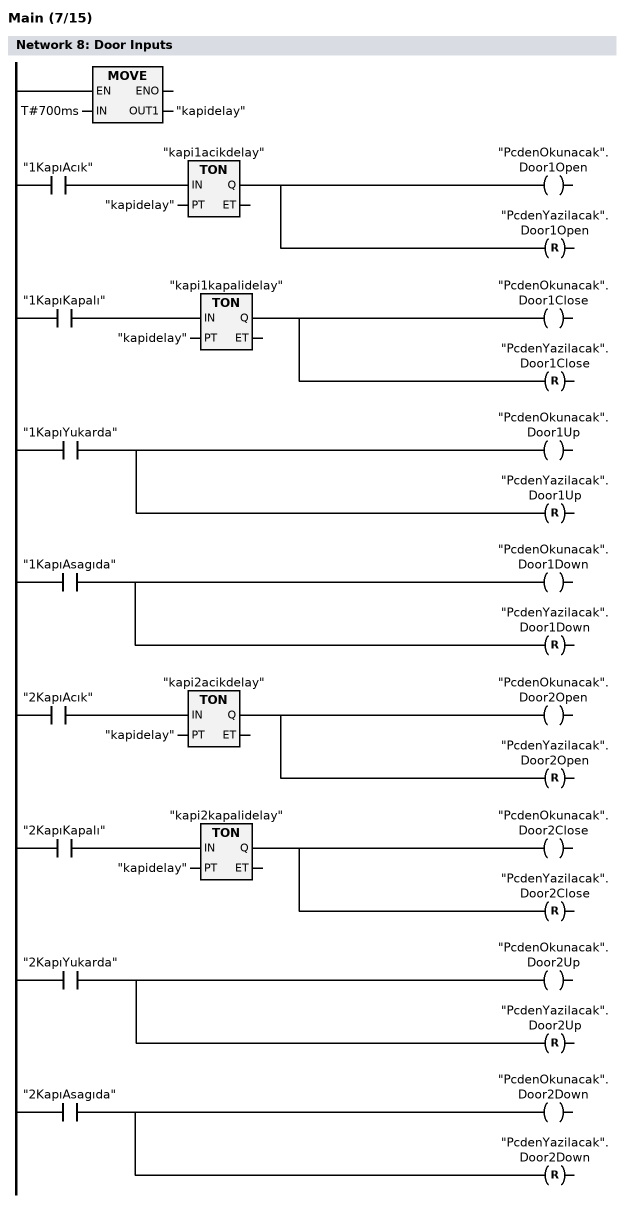
   "kapidelay" := T#700ms;
   "kapi1acikdelay".TON(IN := "1KapıAcık", PT := "kapidelay");
   "PcdenOkunacak".Door1Open := "kapi1acikdelay".Q;
   IF "kapi1acikdelay".Q THEN "PcdenYazilacak".Door1Open := FALSE; END_IF;
   "kapi1kapalidelay".TON(IN := "1KapıKapalı", PT := "kapidelay");
   "PcdenOkunacak".Door1Close := "kapi1kapalidelay".Q;
   IF "kapi1kapalidelay".Q THEN "PcdenYazilacak".Door1Close := FALSE; END_IF;
   "PcdenOkunacak".Door1Up := "1KapıYukarda";
   IF "1KapıYukarda" THEN "PcdenYazilacak".Door1Up := FALSE; END_IF;
   "PcdenOkunacak".Door1Down := "1KapıAsagıda";
   IF "1KapıAsagıda" THEN "PcdenYazilacak".Door1Down := FALSE; END_IF;
   "kapi2acikdelay".TON(IN := "2KapıAcık", PT := "kapidelay");
   "PcdenOkunacak".Door2Open := "kapi2acikdelay".Q;
   IF "kapi2acikdelay".Q THEN "PcdenYazilacak".Door2Open := FALSE; END_IF;
   "kapi2kapalidelay".TON(IN := "2KapıKapalı", PT := "kapidelay");
   "PcdenOkunacak".Door2Close := "kapi2kapalidelay".Q;
   IF "kapi2kapalidelay".Q THEN "PcdenYazilacak".Door2Close := FALSE; END_IF;
   "PcdenOkunacak".Door2Up := "2KapıYukarda";
   IF "2KapıYukarda" THEN "PcdenYazilacak".Door2Up := FALSE; END_IF;
   "PcdenOkunacak".Door2Down := "2KapıAsagıda";
   IF "2KapıAsagıda" THEN "PcdenYazilacak".Door2Down := FALSE; END_IF;
END_REGION

REGION Network 9: Door 1 Outputs
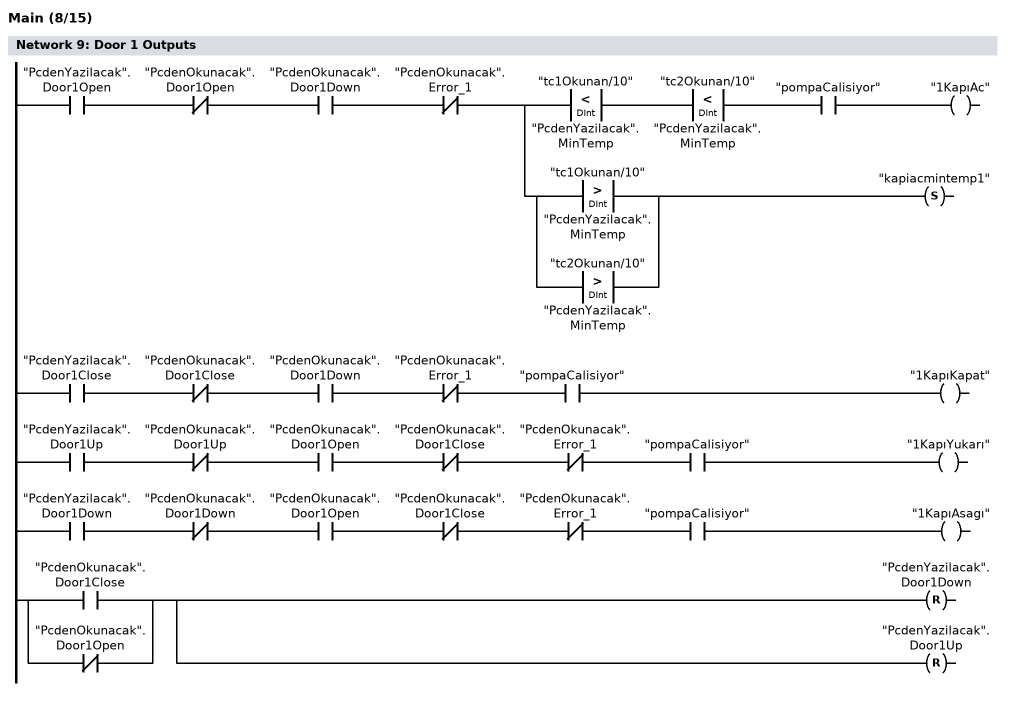
   RUNG wire#powerrail
      Contact( "PcdenYazilacak".Door1Open )
      I_Contact( "PcdenOkunacak".Door1Open )
      Contact( "PcdenOkunacak".Door1Down )
      I_Contact( "PcdenOkunacak".Error_1 )
      wire#w1
      { S7_Templates := "SrcType := DInt" } LT_Contact(in1 := "tc1Okunan/10", in2 := "PcdenYazilacak".MinTemp)
      { S7_Templates := "SrcType := DInt" } LT_Contact(in1 := "tc2Okunan/10", in2 := "PcdenYazilacak".MinTemp)
      Contact( "pompaCalisiyor" )
      Coil( "1KapıAc" )
   END_RUNG
   RUNG wire#w1
      { S7_Templates := "SrcType := DInt" } GT_Contact(in1 := "tc1Okunan/10", in2 := "PcdenYazilacak".MinTemp)
      wire#w2
      S_Coil( "kapiacmintemp1" )
   END_RUNG
   RUNG wire#w1
      { S7_Templates := "SrcType := DInt" } GT_Contact(in1 := "tc2Okunan/10", in2 := "PcdenYazilacak".MinTemp)
   END_RUNG wire#w2
   RUNG wire#powerrail
      Contact( "PcdenYazilacak".Door1Close )
      I_Contact( "PcdenOkunacak".Door1Close )
      Contact( "PcdenOkunacak".Door1Down )
      I_Contact( "PcdenOkunacak".Error_1 )
      Contact( "pompaCalisiyor" )
      Coil( "1KapıKapat" )
   END_RUNG
   RUNG wire#powerrail
      Contact( "PcdenYazilacak".Door1Up )
      I_Contact( "PcdenOkunacak".Door1Up )
      Contact( "PcdenOkunacak".Door1Open )
      I_Contact( "PcdenOkunacak".Door1Close )
      I_Contact( "PcdenOkunacak".Error_1 )
      Contact( "pompaCalisiyor" )
      Coil( "1KapıYukarı" )
   END_RUNG
   RUNG wire#powerrail
      Contact( "PcdenYazilacak".Door1Down )
      I_Contact( "PcdenOkunacak".Door1Down )
      Contact( "PcdenOkunacak".Door1Open )
      I_Contact( "PcdenOkunacak".Door1Close )
      I_Contact( "PcdenOkunacak".Error_1 )
      Contact( "pompaCalisiyor" )
      Coil( "1KapıAsagı" )
   END_RUNG
   RUNG wire#powerrail
      Contact( "PcdenOkunacak".Door1Close )
      wire#w3
      R_Coil( "PcdenYazilacak".Door1Down )
   END_RUNG
   RUNG wire#powerrail
      I_Contact( "PcdenOkunacak".Door1Open )
   END_RUNG wire#w3
   RUNG wire#w3
      R_Coil( "PcdenYazilacak".Door1Up )
   END_RUNG
   // the same network as SCL:
   #_w1 := "PcdenYazilacak".Door1Open AND NOT "PcdenOkunacak".Door1Open AND "PcdenOkunacak".Door1Down AND NOT "PcdenOkunacak".Error_1;
   "1KapıAc" := #_w1 AND ("tc1Okunan/10" < "PcdenYazilacak".MinTemp) AND ("tc2Okunan/10" < "PcdenYazilacak".MinTemp) AND "pompaCalisiyor";
   IF #_w1 AND (("tc1Okunan/10" > "PcdenYazilacak".MinTemp) OR ("tc2Okunan/10" > "PcdenYazilacak".MinTemp)) THEN
       "kapiacmintemp1" := TRUE;
   END_IF;
   "1KapıKapat" := "PcdenYazilacak".Door1Close AND NOT "PcdenOkunacak".Door1Close AND "PcdenOkunacak".Door1Down AND NOT "PcdenOkunacak".Error_1 AND "pompaCalisiyor";
   "1KapıYukarı" := "PcdenYazilacak".Door1Up AND NOT "PcdenOkunacak".Door1Up AND "PcdenOkunacak".Door1Open AND NOT "PcdenOkunacak".Door1Close AND NOT "PcdenOkunacak".Error_1 AND "pompaCalisiyor";
   "1KapıAsagı" := "PcdenYazilacak".Door1Down AND NOT "PcdenOkunacak".Door1Down AND "PcdenOkunacak".Door1Open AND NOT "PcdenOkunacak".Door1Close AND NOT "PcdenOkunacak".Error_1 AND "pompaCalisiyor";
   IF "PcdenOkunacak".Door1Close OR NOT "PcdenOkunacak".Door1Open THEN
       "PcdenYazilacak".Door1Down := FALSE;
       "PcdenYazilacak".Door1Up := FALSE;
   END_IF;
END_REGION

REGION Network 10: Door 2 Outputs
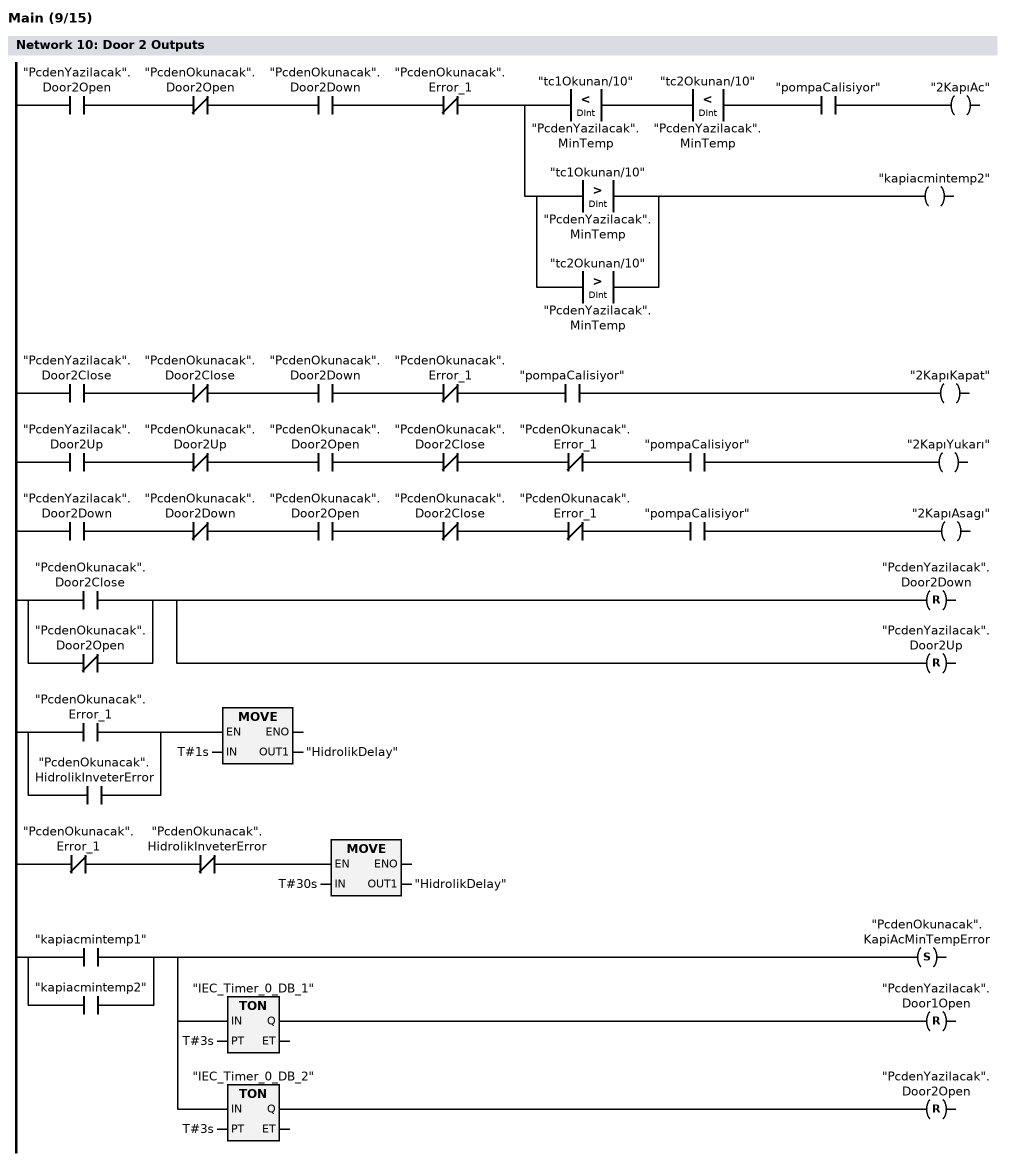
   #_w1 := "PcdenYazilacak".Door2Open AND NOT "PcdenOkunacak".Door2Open AND "PcdenOkunacak".Door2Down AND NOT "PcdenOkunacak".Error_1;
   "2KapıAc" := #_w1 AND ("tc1Okunan/10" < "PcdenYazilacak".MinTemp) AND ("tc2Okunan/10" < "PcdenYazilacak".MinTemp) AND "pompaCalisiyor";
   "kapiacmintemp2" := #_w1 AND (("tc1Okunan/10" > "PcdenYazilacak".MinTemp) OR ("tc2Okunan/10" > "PcdenYazilacak".MinTemp));
   "2KapıKapat" := "PcdenYazilacak".Door2Close AND NOT "PcdenOkunacak".Door2Close AND "PcdenOkunacak".Door2Down AND NOT "PcdenOkunacak".Error_1 AND "pompaCalisiyor";
   "2KapıYukarı" := "PcdenYazilacak".Door2Up AND NOT "PcdenOkunacak".Door2Up AND "PcdenOkunacak".Door2Open AND NOT "PcdenOkunacak".Door2Close AND NOT "PcdenOkunacak".Error_1 AND "pompaCalisiyor";
   "2KapıAsagı" := "PcdenYazilacak".Door2Down AND NOT "PcdenOkunacak".Door2Down AND "PcdenOkunacak".Door2Open AND NOT "PcdenOkunacak".Door2Close AND NOT "PcdenOkunacak".Error_1 AND "pompaCalisiyor";
   IF "PcdenOkunacak".Door2Close OR NOT "PcdenOkunacak".Door2Open THEN
       "PcdenYazilacak".Door2Down := FALSE;
       "PcdenYazilacak".Door2Up := FALSE;
   END_IF;
   IF "PcdenOkunacak".Error_1 OR "PcdenOkunacak".HidrolikInveterError THEN "HidrolikDelay" := T#1s; END_IF;
   IF NOT "PcdenOkunacak".Error_1 AND NOT "PcdenOkunacak".HidrolikInveterError THEN
       "HidrolikDelay" := T#30s;
   END_IF;
   #_w2 := "kapiacmintemp1" OR "kapiacmintemp2";
   IF #_w2 THEN "PcdenOkunacak".KapiAcMinTempError := TRUE; END_IF;
   "IEC_Timer_0_DB_1".TON(IN := #_w2, PT := T#3s);
   IF "IEC_Timer_0_DB_1".Q THEN "PcdenYazilacak".Door1Open := FALSE; END_IF;
   "IEC_Timer_0_DB_2".TON(IN := #_w2, PT := T#3s);
   IF "IEC_Timer_0_DB_2".Q THEN "PcdenYazilacak".Door2Open := FALSE; END_IF;
END_REGION

REGION Network 11: Hidrolik Pompa
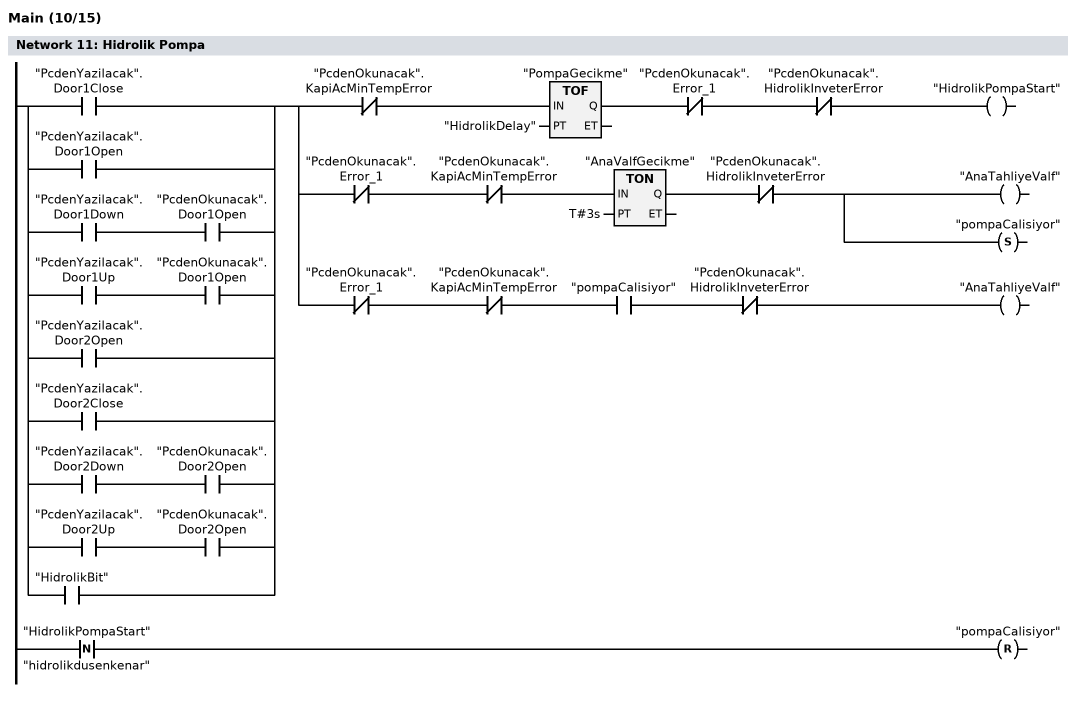
   #_w1 := "PcdenYazilacak".Door1Close OR "PcdenYazilacak".Door1Open OR ("PcdenYazilacak".Door1Down AND "PcdenOkunacak".Door1Open) OR ("PcdenYazilacak".Door1Up AND "PcdenOkunacak".Door1Open) OR "PcdenYazilacak".Door2Open OR "PcdenYazilacak".Door2Close OR ("PcdenYazilacak".Door2Down AND "PcdenOkunacak".Door2Open) OR ("PcdenYazilacak".Door2Up AND "PcdenOkunacak".Door2Open) OR "HidrolikBit";
   "PompaGecikme".TOF(IN := #_w1 AND NOT "PcdenOkunacak".KapiAcMinTempError, PT := "HidrolikDelay");
   "HidrolikPompaStart" := "PompaGecikme".Q AND NOT "PcdenOkunacak".Error_1 AND NOT "PcdenOkunacak".HidrolikInveterError;
   "AnaValfGecikme".TON(IN := #_w1 AND NOT "PcdenOkunacak".Error_1 AND NOT "PcdenOkunacak".KapiAcMinTempError,
                        PT := T#3s);
   "AnaTahliyeValf" := "AnaValfGecikme".Q AND NOT "PcdenOkunacak".HidrolikInveterError;
   IF "AnaTahliyeValf" THEN "pompaCalisiyor" := TRUE; END_IF;
   "AnaTahliyeValf" := #_w1 AND NOT "PcdenOkunacak".Error_1 AND NOT "PcdenOkunacak".KapiAcMinTempError AND "pompaCalisiyor" AND NOT "PcdenOkunacak".HidrolikInveterError;
   #_w2 := NOT "HidrolikPompaStart" AND "hidrolikdusenkenar";   // falling edge of "HidrolikPompaStart"
   "hidrolikdusenkenar" := "HidrolikPompaStart";
   IF #_w2 THEN "pompaCalisiyor" := FALSE; END_IF;
END_REGION

REGION Network 12: Communication
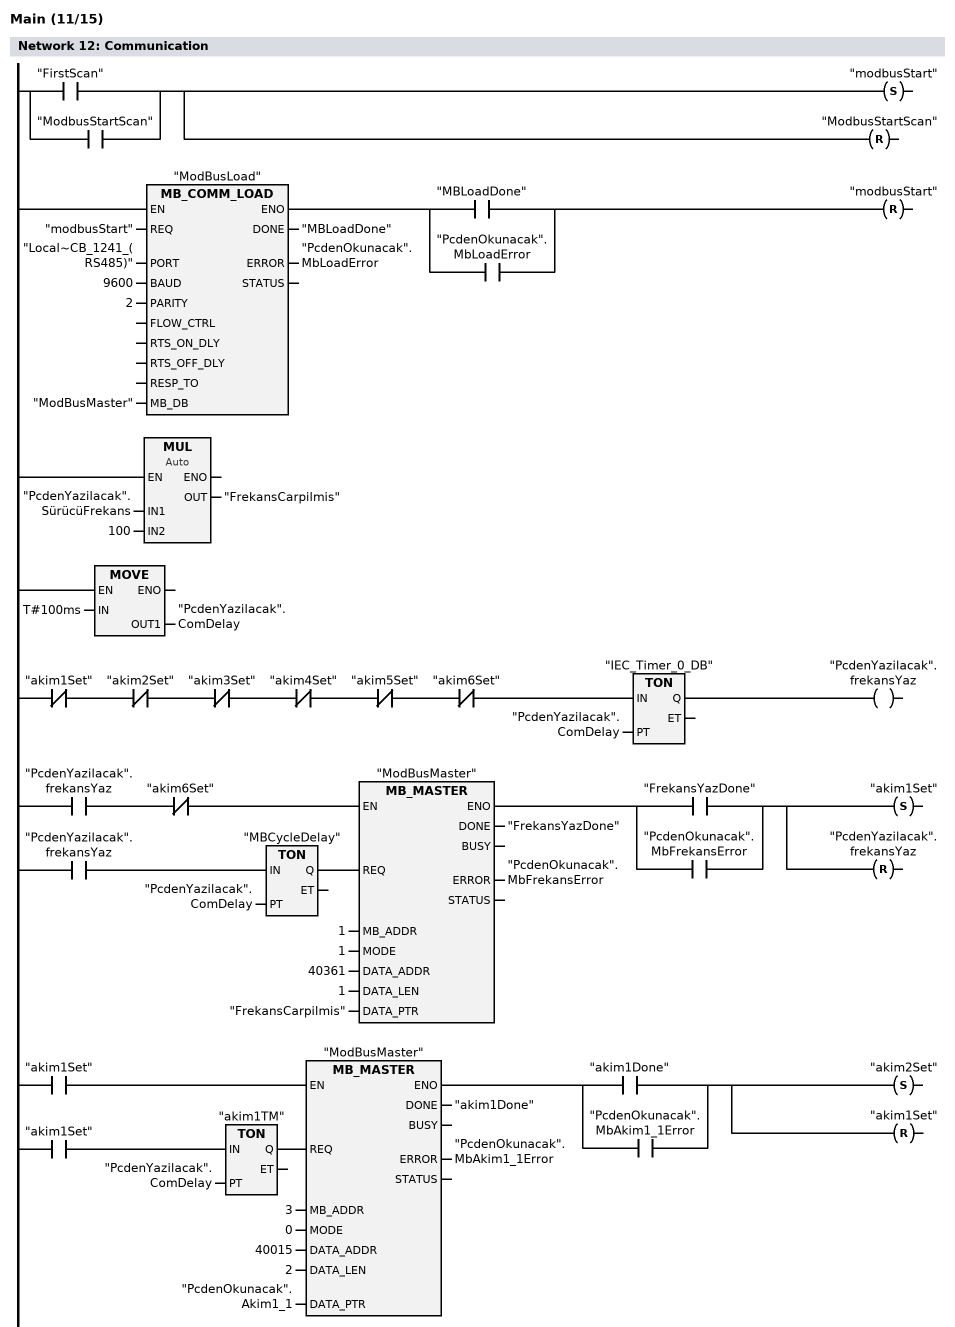
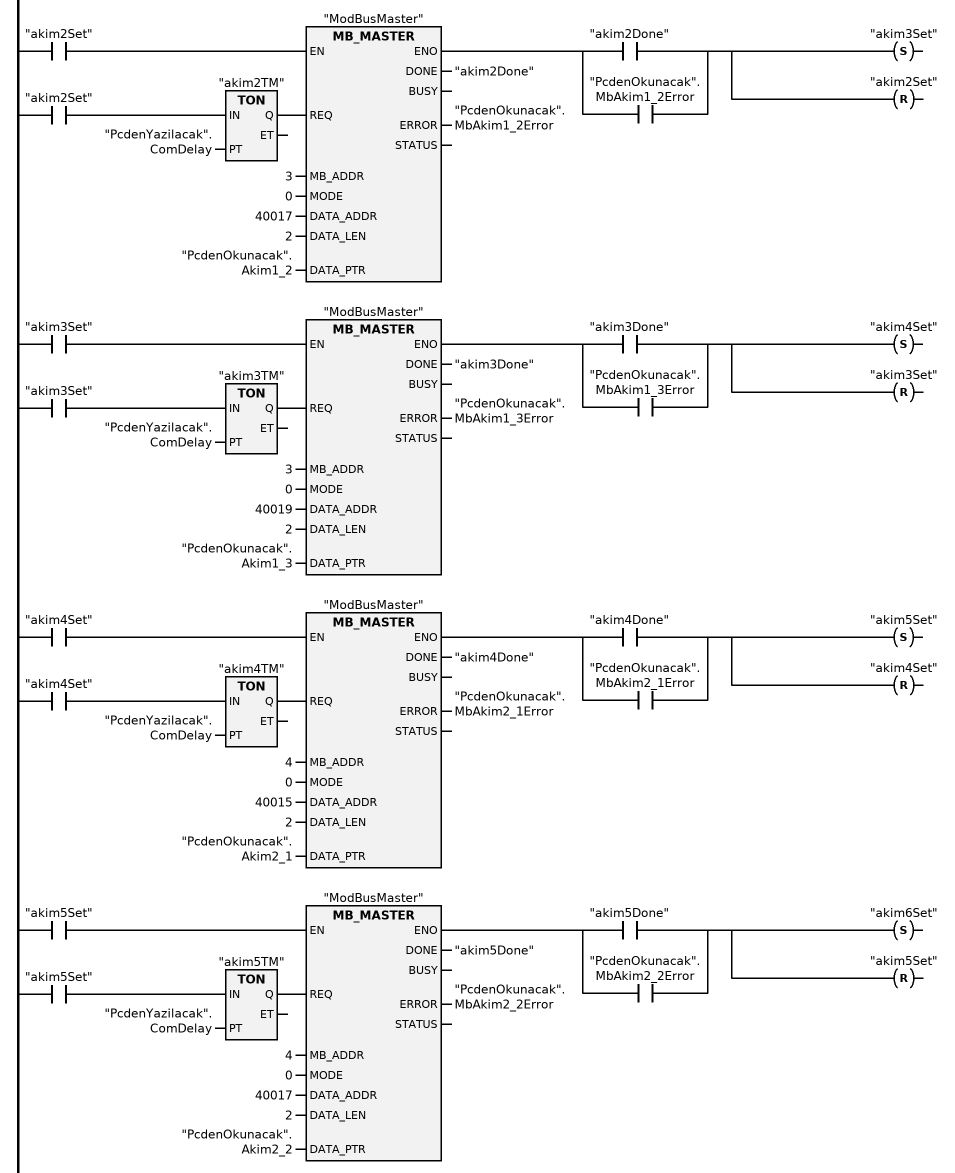
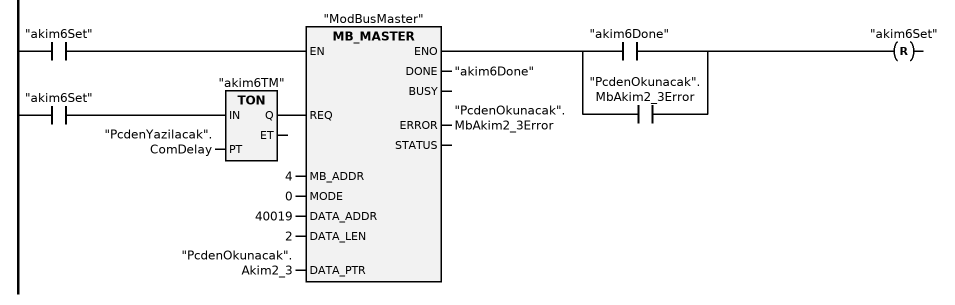
   // ENO of a box is taken as its EN; it also drops when the box reports an error
   IF "FirstScan" OR "ModbusStartScan" THEN
       "modbusStart" := TRUE;
       "ModbusStartScan" := FALSE;
   END_IF;
   "ModBusLoad"(REQ := "modbusStart",   // MB_COMM_LOAD
                PORT := "Local~CB_1241_(RS485)",
                BAUD := 9600,
                PARITY := 2,
                MB_DB := "ModBusMaster",
                DONE => "MBLoadDone",
                ERROR => "PcdenOkunacak".MbLoadError);
   IF "MBLoadDone" OR "PcdenOkunacak".MbLoadError THEN "modbusStart" := FALSE; END_IF;
   "FrekansCarpilmis" := "PcdenYazilacak".SürücüFrekans * 100;
   "PcdenYazilacak".ComDelay := T#100ms;
   "IEC_Timer_0_DB".TON(IN := NOT "akim1Set" AND NOT "akim2Set" AND NOT "akim3Set" AND NOT "akim4Set" AND NOT "akim5Set" AND NOT "akim6Set",
                        PT := "PcdenYazilacak".ComDelay);
   "PcdenYazilacak".frekansYaz := "IEC_Timer_0_DB".Q;
   #_w1 := "PcdenYazilacak".frekansYaz AND NOT "akim6Set";
   "MBCycleDelay".TON(IN := "PcdenYazilacak".frekansYaz, PT := "PcdenYazilacak".ComDelay);
   IF #_w1 THEN
       "ModBusMaster"(REQ := "MBCycleDelay".Q,   // MB_MASTER
                      MB_ADDR := 1,
                      MODE := 1,
                      DATA_ADDR := 40361,
                      DATA_LEN := 1,
                      DATA_PTR := "FrekansCarpilmis",
                      DONE => "FrekansYazDone",
                      ERROR => "PcdenOkunacak".MbFrekansError);
   END_IF;
   IF #_w1 AND ("FrekansYazDone" OR "PcdenOkunacak".MbFrekansError) THEN
       "akim1Set" := TRUE;
       "PcdenYazilacak".frekansYaz := FALSE;
   END_IF;
   "akim1TM".TON(IN := "akim1Set", PT := "PcdenYazilacak".ComDelay);
   #_w2 := "akim1Set";
   IF #_w2 THEN
       "ModBusMaster"(REQ := "akim1TM".Q,   // MB_MASTER
                      MB_ADDR := 3,
                      MODE := 0,
                      DATA_ADDR := 40015,
                      DATA_LEN := 2,
                      DATA_PTR := "PcdenOkunacak".Akim1_1,
                      DONE => "akim1Done",
                      ERROR => "PcdenOkunacak".MbAkim1_1Error);
   END_IF;
   IF #_w2 AND ("akim1Done" OR "PcdenOkunacak".MbAkim1_1Error) THEN
       "akim2Set" := TRUE;
       "akim1Set" := FALSE;
   END_IF;
   "akim2TM".TON(IN := "akim2Set", PT := "PcdenYazilacak".ComDelay);
   #_w3 := "akim2Set";
   IF #_w3 THEN
       "ModBusMaster"(REQ := "akim2TM".Q,   // MB_MASTER
                      MB_ADDR := 3,
                      MODE := 0,
                      DATA_ADDR := 40017,
                      DATA_LEN := 2,
                      DATA_PTR := "PcdenOkunacak".Akim1_2,
                      DONE => "akim2Done",
                      ERROR => "PcdenOkunacak".MbAkim1_2Error);
   END_IF;
   IF #_w3 AND ("akim2Done" OR "PcdenOkunacak".MbAkim1_2Error) THEN
       "akim3Set" := TRUE;
       "akim2Set" := FALSE;
   END_IF;
   "akim3TM".TON(IN := "akim3Set", PT := "PcdenYazilacak".ComDelay);
   #_w4 := "akim3Set";
   IF #_w4 THEN
       "ModBusMaster"(REQ := "akim3TM".Q,   // MB_MASTER
                      MB_ADDR := 3,
                      MODE := 0,
                      DATA_ADDR := 40019,
                      DATA_LEN := 2,
                      DATA_PTR := "PcdenOkunacak".Akim1_3,
                      DONE => "akim3Done",
                      ERROR => "PcdenOkunacak".MbAkim1_3Error);
   END_IF;
   IF #_w4 AND ("akim3Done" OR "PcdenOkunacak".MbAkim1_3Error) THEN
       "akim4Set" := TRUE;
       "akim3Set" := FALSE;
   END_IF;
   "akim4TM".TON(IN := "akim4Set", PT := "PcdenYazilacak".ComDelay);
   #_w5 := "akim4Set";
   IF #_w5 THEN
       "ModBusMaster"(REQ := "akim4TM".Q,   // MB_MASTER
                      MB_ADDR := 4,
                      MODE := 0,
                      DATA_ADDR := 40015,
                      DATA_LEN := 2,
                      DATA_PTR := "PcdenOkunacak".Akim2_1,
                      DONE => "akim4Done",
                      ERROR => "PcdenOkunacak".MbAkim2_1Error);
   END_IF;
   IF #_w5 AND ("akim4Done" OR "PcdenOkunacak".MbAkim2_1Error) THEN
       "akim5Set" := TRUE;
       "akim4Set" := FALSE;
   END_IF;
   "akim5TM".TON(IN := "akim5Set", PT := "PcdenYazilacak".ComDelay);
   #_w6 := "akim5Set";
   IF #_w6 THEN
       "ModBusMaster"(REQ := "akim5TM".Q,   // MB_MASTER
                      MB_ADDR := 4,
                      MODE := 0,
                      DATA_ADDR := 40017,
                      DATA_LEN := 2,
                      DATA_PTR := "PcdenOkunacak".Akim2_2,
                      DONE => "akim5Done",
                      ERROR => "PcdenOkunacak".MbAkim2_2Error);
   END_IF;
   IF #_w6 AND ("akim5Done" OR "PcdenOkunacak".MbAkim2_2Error) THEN
       "akim6Set" := TRUE;
       "akim5Set" := FALSE;
   END_IF;
   "akim6TM".TON(IN := "akim6Set", PT := "PcdenYazilacak".ComDelay);
   #_w7 := "akim6Set";
   IF #_w7 THEN
       "ModBusMaster"(REQ := "akim6TM".Q,   // MB_MASTER
                      MB_ADDR := 4,
                      MODE := 0,
                      DATA_ADDR := 40019,
                      DATA_LEN := 2,
                      DATA_PTR := "PcdenOkunacak".Akim2_3,
                      DONE => "akim6Done",
                      ERROR => "PcdenOkunacak".MbAkim2_3Error);
   END_IF;
   IF #_w7 AND ("akim6Done" OR "PcdenOkunacak".MbAkim2_3Error) THEN "akim6Set" := FALSE; END_IF;
END_REGION

REGION Network 13: akim ortalama
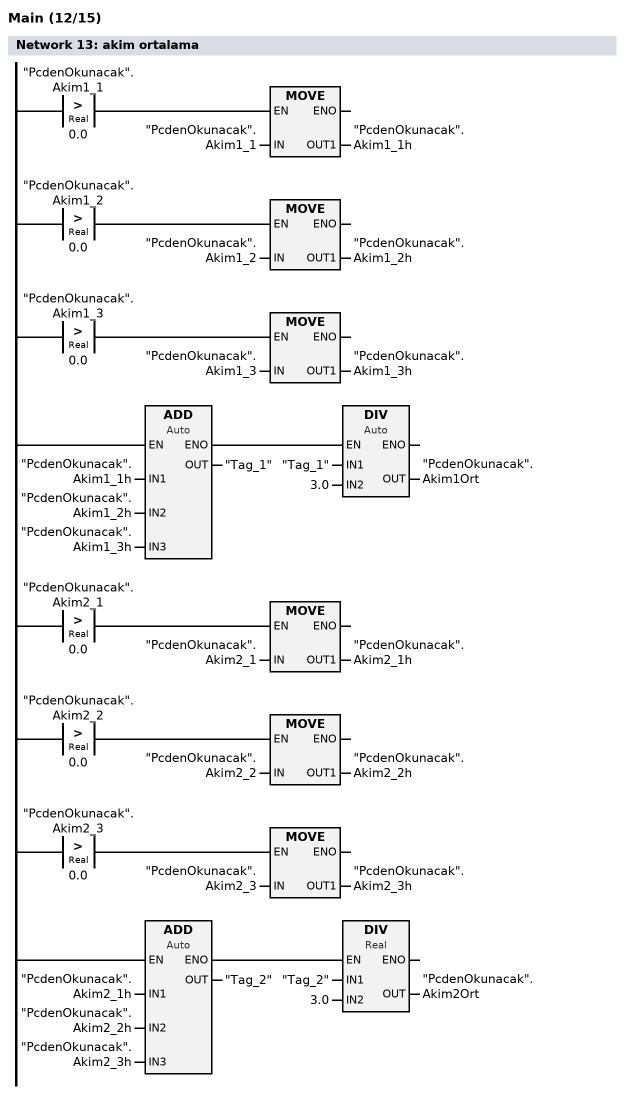
   RUNG wire#powerrail
      { S7_Templates := "SrcType := Real" } GT_Contact(in1 := "PcdenOkunacak".Akim1_1, in2 := 0.0)
      Move(in := "PcdenOkunacak".Akim1_1, out1 => "PcdenOkunacak".Akim1_1h)
   END_RUNG
   RUNG wire#powerrail
      { S7_Templates := "SrcType := Real" } GT_Contact(in1 := "PcdenOkunacak".Akim1_2, in2 := 0.0)
      Move(in := "PcdenOkunacak".Akim1_2, out1 => "PcdenOkunacak".Akim1_2h)
   END_RUNG
   RUNG wire#powerrail
      { S7_Templates := "SrcType := Real" } GT_Contact(in1 := "PcdenOkunacak".Akim1_3, in2 := 0.0)
      Move(in := "PcdenOkunacak".Akim1_3, out1 => "PcdenOkunacak".Akim1_3h)
   END_RUNG
   RUNG wire#powerrail
      Add(in1 := "PcdenOkunacak".Akim1_1h, in2 := "PcdenOkunacak".Akim1_2h, in3 := "PcdenOkunacak".Akim1_3h, out => "Tag_1")
      Div(in1 := "Tag_1", in2 := 3.0, out => "PcdenOkunacak".Akim1Ort)
   END_RUNG
   RUNG wire#powerrail
      { S7_Templates := "SrcType := Real" } GT_Contact(in1 := "PcdenOkunacak".Akim2_1, in2 := 0.0)
      Move(in := "PcdenOkunacak".Akim2_1, out1 => "PcdenOkunacak".Akim2_1h)
   END_RUNG
   RUNG wire#powerrail
      { S7_Templates := "SrcType := Real" } GT_Contact(in1 := "PcdenOkunacak".Akim2_2, in2 := 0.0)
      Move(in := "PcdenOkunacak".Akim2_2, out1 => "PcdenOkunacak".Akim2_2h)
   END_RUNG
   RUNG wire#powerrail
      { S7_Templates := "SrcType := Real" } GT_Contact(in1 := "PcdenOkunacak".Akim2_3, in2 := 0.0)
      Move(in := "PcdenOkunacak".Akim2_3, out1 => "PcdenOkunacak".Akim2_3h)
   END_RUNG
   RUNG wire#powerrail
      Add(in1 := "PcdenOkunacak".Akim2_1h, in2 := "PcdenOkunacak".Akim2_2h, in3 := "PcdenOkunacak".Akim2_3h, out => "Tag_2")
      { S7_Templates := "SrcType := Real" } Div(in1 := "Tag_2", in2 := 3.0, out => "PcdenOkunacak".Akim2Ort)
   END_RUNG
   // the same network as SCL:
   IF "PcdenOkunacak".Akim1_1 > 0.0 THEN "PcdenOkunacak".Akim1_1h := "PcdenOkunacak".Akim1_1; END_IF;
   IF "PcdenOkunacak".Akim1_2 > 0.0 THEN "PcdenOkunacak".Akim1_2h := "PcdenOkunacak".Akim1_2; END_IF;
   IF "PcdenOkunacak".Akim1_3 > 0.0 THEN "PcdenOkunacak".Akim1_3h := "PcdenOkunacak".Akim1_3; END_IF;
   "Tag_1" := "PcdenOkunacak".Akim1_1h + "PcdenOkunacak".Akim1_2h + "PcdenOkunacak".Akim1_3h;
   "PcdenOkunacak".Akim1Ort := "Tag_1" / 3.0;
   IF "PcdenOkunacak".Akim2_1 > 0.0 THEN "PcdenOkunacak".Akim2_1h := "PcdenOkunacak".Akim2_1; END_IF;
   IF "PcdenOkunacak".Akim2_2 > 0.0 THEN "PcdenOkunacak".Akim2_2h := "PcdenOkunacak".Akim2_2; END_IF;
   IF "PcdenOkunacak".Akim2_3 > 0.0 THEN "PcdenOkunacak".Akim2_3h := "PcdenOkunacak".Akim2_3; END_IF;
   "Tag_2" := "PcdenOkunacak".Akim2_1h + "PcdenOkunacak".Akim2_2h + "PcdenOkunacak".Akim2_3h;
   "PcdenOkunacak".Akim2Ort := "Tag_2" / 3.0;
END_REGION

REGION Network 14
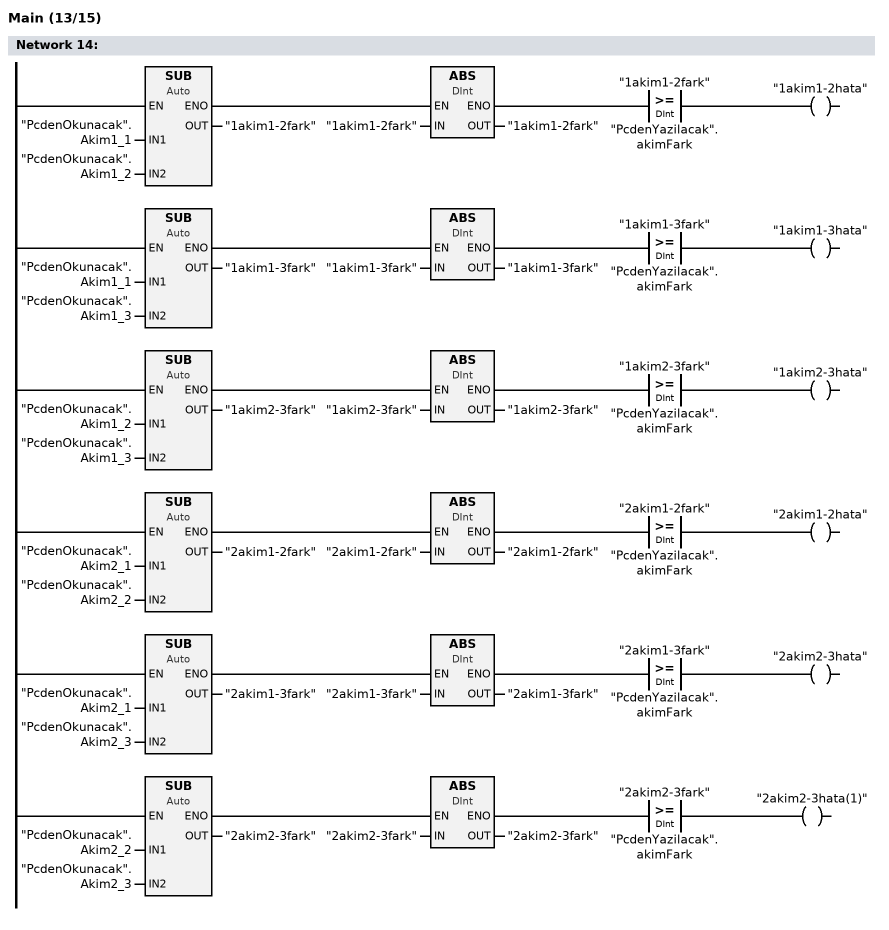
   RUNG wire#powerrail
      Sub(in1 := "PcdenOkunacak".Akim1_1, in2 := "PcdenOkunacak".Akim1_2, out => "1akim1-2fark")
      { S7_Templates := "SrcType := DInt" } Abs(in := "1akim1-2fark", out => "1akim1-2fark")
      { S7_Templates := "SrcType := DInt" } GE_Contact(in1 := "1akim1-2fark", in2 := "PcdenYazilacak".akimFark)
      Coil( "1akim1-2hata" )
   END_RUNG
   RUNG wire#powerrail
      Sub(in1 := "PcdenOkunacak".Akim1_1, in2 := "PcdenOkunacak".Akim1_3, out => "1akim1-3fark")
      { S7_Templates := "SrcType := DInt" } Abs(in := "1akim1-3fark", out => "1akim1-3fark")
      { S7_Templates := "SrcType := DInt" } GE_Contact(in1 := "1akim1-3fark", in2 := "PcdenYazilacak".akimFark)
      Coil( "1akim1-3hata" )
   END_RUNG
   RUNG wire#powerrail
      Sub(in1 := "PcdenOkunacak".Akim1_2, in2 := "PcdenOkunacak".Akim1_3, out => "1akim2-3fark")
      { S7_Templates := "SrcType := DInt" } Abs(in := "1akim2-3fark", out => "1akim2-3fark")
      { S7_Templates := "SrcType := DInt" } GE_Contact(in1 := "1akim2-3fark", in2 := "PcdenYazilacak".akimFark)
      Coil( "1akim2-3hata" )
   END_RUNG
   RUNG wire#powerrail
      Sub(in1 := "PcdenOkunacak".Akim2_1, in2 := "PcdenOkunacak".Akim2_2, out => "2akim1-2fark")
      { S7_Templates := "SrcType := DInt" } Abs(in := "2akim1-2fark", out => "2akim1-2fark")
      { S7_Templates := "SrcType := DInt" } GE_Contact(in1 := "2akim1-2fark", in2 := "PcdenYazilacak".akimFark)
      Coil( "2akim1-2hata" )
   END_RUNG
   RUNG wire#powerrail
      Sub(in1 := "PcdenOkunacak".Akim2_1, in2 := "PcdenOkunacak".Akim2_3, out => "2akim1-3fark")
      { S7_Templates := "SrcType := DInt" } Abs(in := "2akim1-3fark", out => "2akim1-3fark")
      { S7_Templates := "SrcType := DInt" } GE_Contact(in1 := "2akim1-3fark", in2 := "PcdenYazilacak".akimFark)
      Coil( "2akim2-3hata" )
   END_RUNG
   RUNG wire#powerrail
      Sub(in1 := "PcdenOkunacak".Akim2_2, in2 := "PcdenOkunacak".Akim2_3, out => "2akim2-3fark")
      { S7_Templates := "SrcType := DInt" } Abs(in := "2akim2-3fark", out => "2akim2-3fark")
      { S7_Templates := "SrcType := DInt" } GE_Contact(in1 := "2akim2-3fark", in2 := "PcdenYazilacak".akimFark)
      Coil( "2akim2-3hata(1)" )
   END_RUNG
   // the same network as SCL:
   "1akim1-2fark" := "PcdenOkunacak".Akim1_1 - "PcdenOkunacak".Akim1_2;
   "1akim1-2fark" := ABS("1akim1-2fark");
   "1akim1-2hata" := "1akim1-2fark" >= "PcdenYazilacak".akimFark;
   "1akim1-3fark" := "PcdenOkunacak".Akim1_1 - "PcdenOkunacak".Akim1_3;
   "1akim1-3fark" := ABS("1akim1-3fark");
   "1akim1-3hata" := "1akim1-3fark" >= "PcdenYazilacak".akimFark;
   "1akim2-3fark" := "PcdenOkunacak".Akim1_2 - "PcdenOkunacak".Akim1_3;
   "1akim2-3fark" := ABS("1akim2-3fark");
   "1akim2-3hata" := "1akim2-3fark" >= "PcdenYazilacak".akimFark;
   "2akim1-2fark" := "PcdenOkunacak".Akim2_1 - "PcdenOkunacak".Akim2_2;
   "2akim1-2fark" := ABS("2akim1-2fark");
   "2akim1-2hata" := "2akim1-2fark" >= "PcdenYazilacak".akimFark;
   "2akim1-3fark" := "PcdenOkunacak".Akim2_1 - "PcdenOkunacak".Akim2_3;
   "2akim1-3fark" := ABS("2akim1-3fark");
   "2akim2-3hata" := "2akim1-3fark" >= "PcdenYazilacak".akimFark;
   "2akim2-3fark" := "PcdenOkunacak".Akim2_2 - "PcdenOkunacak".Akim2_3;
   "2akim2-3fark" := ABS("2akim2-3fark");
   "2akim2-3hata(1)" := "2akim2-3fark" >= "PcdenYazilacak".akimFark;
END_REGION

REGION Network 15: Damper Set
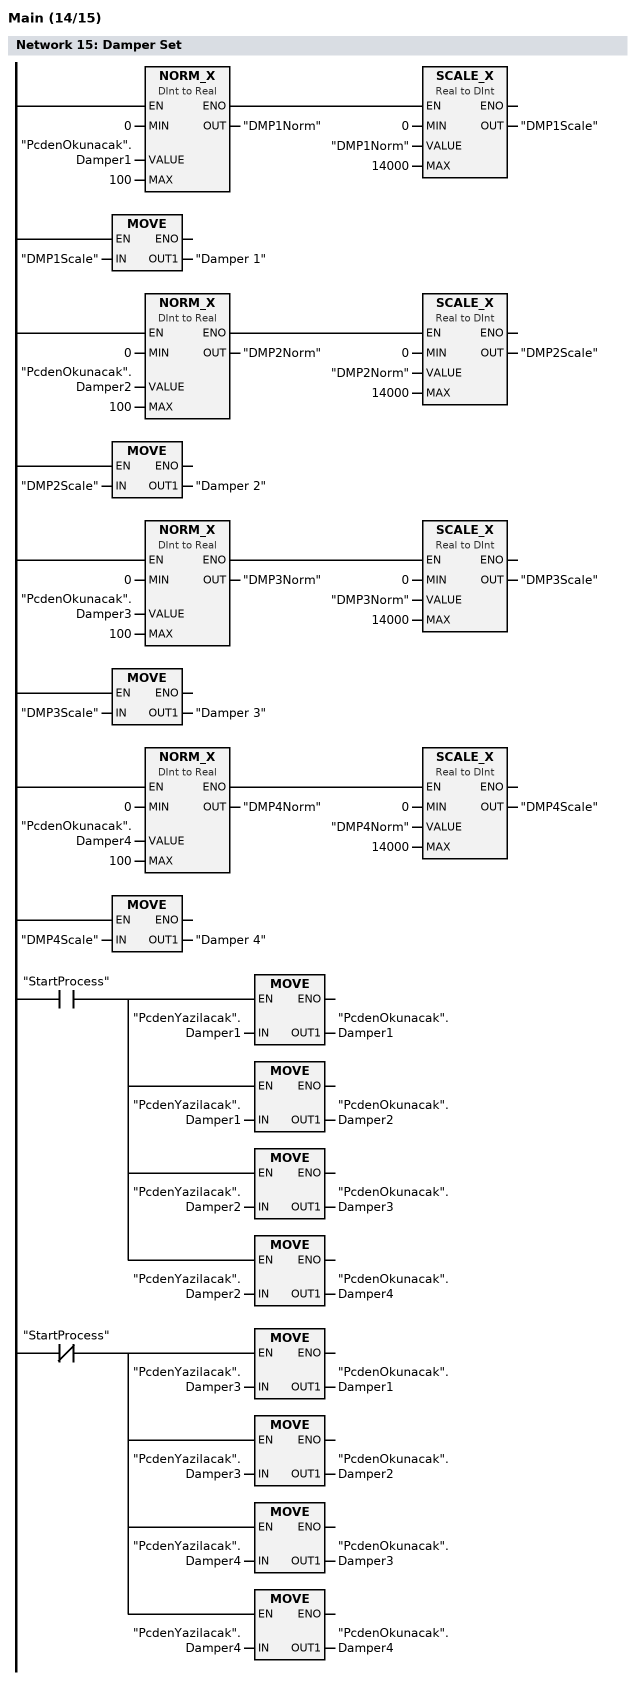
   RUNG wire#powerrail
      { S7_Templates := "[SrcType := DInt, DestType := Real]" } Normalize(min := 0, value := "PcdenOkunacak".Damper1, max := 100, out => "DMP1Norm")
      { S7_Templates := "[SrcType := Real, DestType := DInt]" } Scale(min := 0, value := "DMP1Norm", max := 14000, out => "DMP1Scale")
   END_RUNG
   RUNG wire#powerrail
      Move(in := "DMP1Scale", out1 => "Damper 1")
   END_RUNG
   RUNG wire#powerrail
      { S7_Templates := "[SrcType := DInt, DestType := Real]" } Normalize(min := 0, value := "PcdenOkunacak".Damper2, max := 100, out => "DMP2Norm")
      { S7_Templates := "[SrcType := Real, DestType := DInt]" } Scale(min := 0, value := "DMP2Norm", max := 14000, out => "DMP2Scale")
   END_RUNG
   RUNG wire#powerrail
      Move(in := "DMP2Scale", out1 => "Damper 2")
   END_RUNG
   RUNG wire#powerrail
      { S7_Templates := "[SrcType := DInt, DestType := Real]" } Normalize(min := 0, value := "PcdenOkunacak".Damper3, max := 100, out => "DMP3Norm")
      { S7_Templates := "[SrcType := Real, DestType := DInt]" } Scale(min := 0, value := "DMP3Norm", max := 14000, out => "DMP3Scale")
   END_RUNG
   RUNG wire#powerrail
      Move(in := "DMP3Scale", out1 => "Damper 3")
   END_RUNG
   RUNG wire#powerrail
      { S7_Templates := "[SrcType := DInt, DestType := Real]" } Normalize(min := 0, value := "PcdenOkunacak".Damper4, max := 100, out => "DMP4Norm")
      { S7_Templates := "[SrcType := Real, DestType := DInt]" } Scale(min := 0, value := "DMP4Norm", max := 14000, out => "DMP4Scale")
   END_RUNG
   RUNG wire#powerrail
      Move(in := "DMP4Scale", out1 => "Damper 4")
   END_RUNG
   RUNG wire#powerrail
      Contact( "StartProcess" )
      wire#w1
      Move(in := "PcdenYazilacak".Damper1, out1 => "PcdenOkunacak".Damper1)
   END_RUNG
   RUNG wire#w1
      Move(in := "PcdenYazilacak".Damper1, out1 => "PcdenOkunacak".Damper2)
   END_RUNG
   RUNG wire#w1
      Move(in := "PcdenYazilacak".Damper2, out1 => "PcdenOkunacak".Damper3)
   END_RUNG
   RUNG wire#w1
      Move(in := "PcdenYazilacak".Damper2, out1 => "PcdenOkunacak".Damper4)
   END_RUNG
   RUNG wire#powerrail
      I_Contact( "StartProcess" )
      wire#w2
      Move(in := "PcdenYazilacak".Damper3, out1 => "PcdenOkunacak".Damper1)
   END_RUNG
   RUNG wire#w2
      Move(in := "PcdenYazilacak".Damper3, out1 => "PcdenOkunacak".Damper2)
   END_RUNG
   RUNG wire#w2
      Move(in := "PcdenYazilacak".Damper4, out1 => "PcdenOkunacak".Damper3)
   END_RUNG
   RUNG wire#w2
      Move(in := "PcdenYazilacak".Damper4, out1 => "PcdenOkunacak".Damper4)
   END_RUNG
   // the same network as SCL:
   "DMP1Norm" := NORM_X(MIN := 0, VALUE := "PcdenOkunacak".Damper1, MAX := 100);
   "DMP1Scale" := SCALE_X(MIN := 0, VALUE := "DMP1Norm", MAX := 14000);
   "Damper 1" := "DMP1Scale";
   "DMP2Norm" := NORM_X(MIN := 0, VALUE := "PcdenOkunacak".Damper2, MAX := 100);
   "DMP2Scale" := SCALE_X(MIN := 0, VALUE := "DMP2Norm", MAX := 14000);
   "Damper 2" := "DMP2Scale";
   "DMP3Norm" := NORM_X(MIN := 0, VALUE := "PcdenOkunacak".Damper3, MAX := 100);
   "DMP3Scale" := SCALE_X(MIN := 0, VALUE := "DMP3Norm", MAX := 14000);
   "Damper 3" := "DMP3Scale";
   "DMP4Norm" := NORM_X(MIN := 0, VALUE := "PcdenOkunacak".Damper4, MAX := 100);
   "DMP4Scale" := SCALE_X(MIN := 0, VALUE := "DMP4Norm", MAX := 14000);
   "Damper 4" := "DMP4Scale";
   IF "StartProcess" THEN
       "PcdenOkunacak".Damper1 := "PcdenYazilacak".Damper1;
       "PcdenOkunacak".Damper2 := "PcdenYazilacak".Damper1;
       "PcdenOkunacak".Damper3 := "PcdenYazilacak".Damper2;
       "PcdenOkunacak".Damper4 := "PcdenYazilacak".Damper2;
   END_IF;
   IF NOT "StartProcess" THEN
       "PcdenOkunacak".Damper1 := "PcdenYazilacak".Damper3;
       "PcdenOkunacak".Damper2 := "PcdenYazilacak".Damper3;
       "PcdenOkunacak".Damper3 := "PcdenYazilacak".Damper4;
       "PcdenOkunacak".Damper4 := "PcdenYazilacak".Damper4;
   END_IF;
END_REGION

REGION Network 16
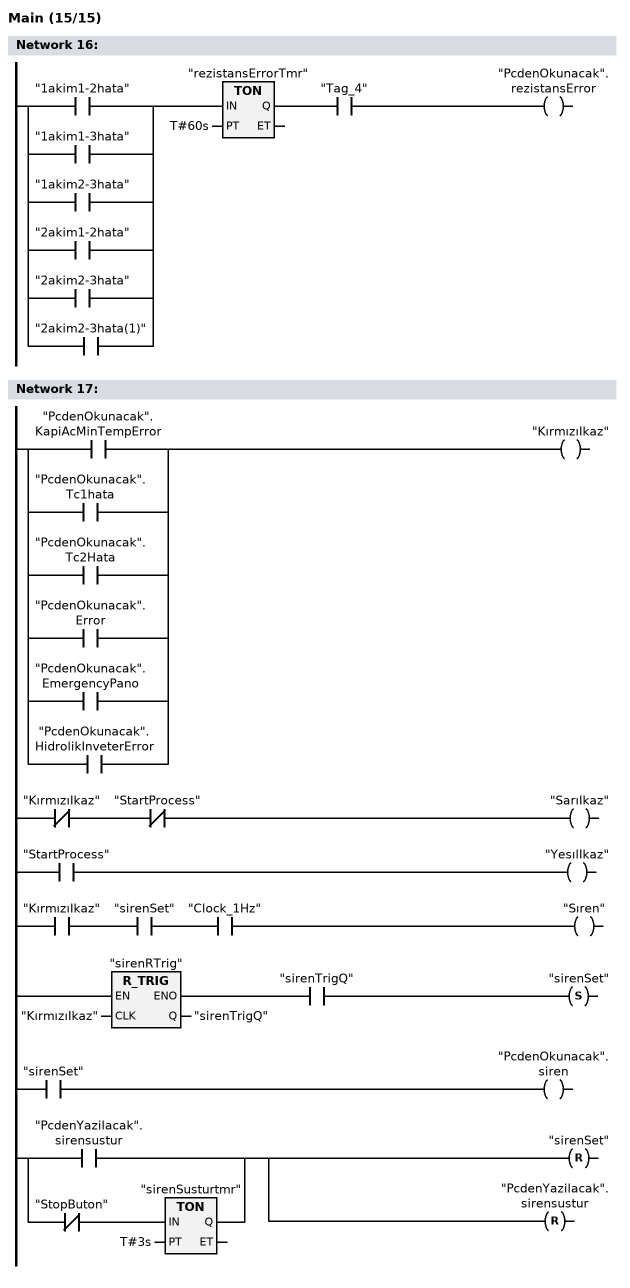
   "rezistansErrorTmr".TON(IN := "1akim1-2hata" OR "1akim1-3hata" OR "1akim2-3hata" OR "2akim1-2hata" OR "2akim2-3hata" OR "2akim2-3hata(1)",
                           PT := T#60s);
   "PcdenOkunacak".rezistansError := "rezistansErrorTmr".Q AND "Tag_4";
END_REGION

REGION Network 17
   // ENO of a box is taken as its EN; it also drops when the box reports an error
   "KırmızıIkaz" := "PcdenOkunacak".KapiAcMinTempError OR "PcdenOkunacak".Tc1hata OR "PcdenOkunacak".Tc2Hata OR "PcdenOkunacak".Error OR "PcdenOkunacak".EmergencyPano OR "PcdenOkunacak".HidrolikInveterError;
   "SarıIkaz" := NOT "KırmızıIkaz" AND NOT "StartProcess";
   "YesılIkaz" := "StartProcess";
   "Sıren" := "KırmızıIkaz" AND "sirenSet" AND "Clock_1Hz";
   "sirenRTrig"(CLK := "KırmızıIkaz", Q => "sirenTrigQ");   // R_TRIG
   IF "sirenTrigQ" THEN "sirenSet" := TRUE; END_IF;
   "PcdenOkunacak".siren := "sirenSet";
   "sirenSusturtmr".TON(IN := NOT "StopButon", PT := T#3s);
   IF "PcdenYazilacak".sirensustur OR "sirenSusturtmr".Q THEN
       "sirenSet" := FALSE;
       "PcdenYazilacak".sirensustur := FALSE;
   END_IF;
END_REGION
END_ORGANIZATION_BLOCK